C07282=1088.457,205.071,426.735,175.963,20.851,153.236
C07283=1088.452,204.821,426.758,175.960,20.850,153.237
C07284=1088.446,204.573,426.782,175.958,20.848,153.237
C07285=1088.441,204.324,426.805,175.955,20.847,153.237
C07286=1088.435,204.076,426.829,175.952,20.845,153.237
C07287=1088.429,203.827,426.853,175.949,20.844,153.237
C07288=1088.424,203.578,426.877,175.946,20.842,153.237
C07289=1088.418,203.329,426.901,175.944,20.841,153.237
C07290=1088.413,203.080,426.924,175.941,20.839,153.237
C07291=1088.407,202.831,426.948,175.938,20.838,153.238
C07292=1088.402,202.582,426.972,175.936,20.837,153.238
C07293=1088.396,202.334,426.995,175.933,20.836,153.238
C07294=1088.391,202.085,427.019,175.929,20.834,153.238
C07295=1088.385,201.836,427.043,175.927,20.833,153.238
C07296=1088.378,201.587,427.066,175.924,20.831,153.238
C07297=1088.373,201.338,427.090,175.922,20.830,153.239
C07298=1088.367,201.089,427.113,175.919,20.829,153.239
C07299=1088.361,200.841,427.137,175.916,20.827,153.239
C07300=1088.356,200.592,427.160,175.914,20.826,153.239
C07301=1088.350,200.344,427.184,175.910,20.824,153.239
C07302=1088.345,200.095,427.207,175.907,20.823,153.239
C07303=1088.340,199.845,427.230,175.905,20.822,153.240
C07304=1088.334,199.597,427.254,175.902,20.820,153.240
C07305=1088.327,199.348,427.277,175.899,20.819,153.240
C07306=1088.322,199.098,427.301,175.897,20.818,153.240
C07307=1088.316,198.850,427.325,175.894,20.816,153.240
C07308=1088.310,198.601,427.348,175.891,20.814,153.240
C07309=1088.305,198.353,427.372,175.888,20.813,153.241
C07310=1088.299,198.104,427.395,175.885,20.812,153.241
C07311=1088.294,197.855,427.418,175.883,20.811,153.241
C07312=1088.289,197.606,427.441,175.880,20.809,153.241
C07313=1088.283,197.357,427.465,175.877,20.808,153.241
C07314=1088.277,197.108,427.488,175.875,20.807,153.241
C07315=1088.272,196.859,427.511,175.872,20.805,153.241
C07316=1088.266,196.611,427.535,175.870,20.804,153.241
C07317=1088.260,196.362,427.558,175.866,20.802,153.242
C07318=1088.254,196.113,427.581,175.863,20.801,153.242
C07319=1088.249,195.864,427.604,175.861,20.800,153.242
C07320=1088.244,195.615,427.627,175.858,20.798,153.242
C07321=1088.238,195.367,427.651,175.856,20.797,153.242
C07322=1088.233,195.118,427.675,175.853,20.795,153.242
C07323=1088.227,194.869,427.698,175.850,20.794,153.243
C07324=1088.221,194.620,427.721,175.848,20.793,153.243
C07325=1088.216,194.371,427.743,175.845,20.791,153.243
C07326=1088.211,194.122,427.767,175.842,20.790,153.243
C07327=1088.205,193.873,427.791,175.840,20.788,153.243
C07328=1088.199,193.624,427.814,175.836,20.787,153.243
C07329=1088.193,193.376,427.837,175.834,20.786,153.243
C07330=1088.187,193.127,427.859,175.831,20.784,153.244
C07331=1088.182,192.877,427.883,175.828,20.783,153.244
C07332=1088.177,192.629,427.906,175.826,20.781,153.244
C07333=1088.171,192.380,427.929,175.823,20.780,153.244
C07334=1088.165,192.103,427.954,175.821,20.778,153.244
C07335=1088.159,191.825,427.981,175.817,20.777,153.244
C07336=1088.153,191.548,428.006,175.814,20.775,153.244
C07337=1088.146,191.270,428.032,175.811,20.774,153.245
C07338=1088.141,191.021,428.055,175.808,20.772,153.245
C07339=1088.135,190.772,428.078,175.806,20.771,153.245
C07340=1088.130,190.523,428.101,175.803,20.769,153.245
C07341=1088.125,190.275,428.124,175.801,20.768,153.245
C07342=1088.119,190.026,428.147,175.798,20.766,153.245
C07343=1088.113,189.777,428.169,175.795,20.765,153.245
C07344=1088.108,189.528,428.193,175.793,20.763,153.245
C07345=1088.102,189.279,428.216,175.790,20.762,153.246
C07346=1088.097,189.030,428.239,175.787,20.761,153.246
C07347=1088.091,188.782,428.261,175.785,20.760,153.246
C07348=1088.086,188.533,428.284,175.782,20.758,153.246
C07349=1088.080,188.284,428.307,175.780,20.757,153.246
C07350=1088.075,188.035,428.330,175.777,20.755,153.246
C07351=1088.070,187.786,428.353,175.775,20.754,153.246
C07352=1088.064,187.537,428.376,175.771,20.752,153.246
C07353=1088.059,187.289,428.399,175.768,20.750,153.247
C07354=1088.053,187.040,428.422,175.766,20.749,153.247
C07355=1088.048,186.790,428.444,175.763,20.748,153.247
C07356=1088.042,186.541,428.467,175.761,20.746,153.247
C07357=1088.037,186.293,428.489,175.758,20.745,153.247
C07358=1088.031,186.044,428.512,175.756,20.743,153.247
C07359=1088.025,185.795,428.535,175.753,20.742,153.247
C07360=1088.021,185.545,428.558,175.750,20.740,153.247
C07361=1088.015,185.297,428.581,175.748,20.739,153.247
C07362=1088.010,185.048,428.604,175.745,20.737,153.248
C07363=1088.003,184.800,428.626,175.743,20.736,153.248
C07364=1087.998,184.550,428.648,175.740,20.735,153.248
C07365=1087.992,184.301,428.671,175.737,20.734,153.248
C07366=1087.986,184.053,428.694,175.735,20.732,153.248
C07367=1087.981,183.803,428.716,175.732,20.731,153.248
C07368=1087.974,183.554,428.739,175.729,20.729,153.248
C07369=1087.969,183.306,428.761,175.727,20.728,153.249
C07370=1087.964,183.057,428.783,175.724,20.727,153.249
C07371=1087.958,182.808,428.806,175.722,20.725,153.249
C07372=1087.952,182.559,428.829,175.719,20.724,153.249
C07373=1087.946,182.310,428.851,175.716,20.722,153.249
C07374=1087.941,182.061,428.874,175.714,20.722,153.249
C07375=1087.935,181.813,428.896,175.711,20.720,153.249
C07376=1087.929,181.563,428.918,175.708,20.719,153.250
C07377=1087.924,181.315,428.941,175.706,20.717,153.250
C07378=1087.918,181.065,428.963,175.703,20.716,153.250
C07379=1087.912,180.816,428.986,175.701,20.714,153.250
C07380=1087.907,180.568,429.008,175.698,20.713,153.250
C07381=1087.901,180.319,429.031,175.695,20.712,153.250
C07382=1087.895,180.070,429.053,175.693,20.710,153.250
C07383=1087.889,179.821,429.075,175.690,20.709,153.251
C07384=1087.884,179.572,429.098,175.687,20.708,153.251
C07385=1087.878,179.323,429.119,175.685,20.706,153.251
C07386=1087.872,179.074,429.142,175.682,20.705,153.251
C07387=1087.867,178.825,429.164,175.680,20.703,153.251
C07388=1087.861,178.576,429.186,175.677,20.702,153.251
C07389=1087.855,178.327,429.209,175.675,20.700,153.251
C07390=1087.850,178.078,429.231,175.672,20.699,153.252
C07391=1087.844,177.829,429.253,175.669,20.698,153.252
C07392=1087.839,177.580,429.275,175.667,20.696,153.252
C07393=1087.833,177.332,429.298,175.664,20.695,153.252
C07394=1087.827,177.082,429.320,175.661,20.694,153.252
C07395=1087.822,176.834,429.342,175.659,20.692,153.252
C07396=1087.816,176.585,429.365,175.656,20.691,153.252
C07397=1087.810,176.335,429.386,175.654,20.689,153.252
C07398=1087.804,176.058,429.411,175.651,20.688,153.252
C07399=1087.798,175.780,429.436,175.648,20.686,153.253
C07400=1087.792,175.502,429.461,175.645,20.684,153.253
C07401=1087.785,175.225,429.485,175.642,20.683,153.253
C07402=1087.780,174.976,429.507,175.640,20.682,153.253
C07403=1087.774,174.727,429.529,175.637,20.680,153.253
C07404=1087.768,174.477,429.551,175.635,20.679,153.253
C07405=1087.763,174.229,429.574,175.632,20.677,153.253
C07406=1087.757,173.980,429.595,175.630,20.676,153.253
C07407=1087.752,173.731,429.617,175.627,20.674,153.254
C07408=1087.746,173.482,429.639,175.624,20.673,153.254
C07409=1087.740,173.233,429.662,175.623,20.672,153.254
C07410=1087.736,172.984,429.684,175.620,20.670,153.254
C07411=1087.729,172.735,429.705,175.617,20.669,153.254
C07412=1087.724,172.486,429.728,175.615,20.668,153.254
C07413=1087.718,172.238,429.750,175.612,20.666,153.254
C07414=1087.713,171.988,429.772,175.610,20.665,153.254
C07415=1087.707,171.740,429.793,175.607,20.663,153.254
C07416=1087.702,171.490,429.815,175.605,20.662,153.255
C07417=1087.696,171.242,429.837,175.602,20.660,153.255
C07418=1087.691,170.992,429.859,175.600,20.658,153.255
C07419=1087.685,170.743,429.881,175.597,20.657,153.255
C07420=1087.679,170.495,429.903,175.594,20.655,153.255
C07421=1087.674,170.245,429.925,175.592,20.654,153.255
C07422=1087.668,169.997,429.947,175.589,20.653,153.255
C07423=1087.663,169.747,429.969,175.587,20.651,153.255
C07424=1087.657,169.499,429.990,175.584,20.650,153.255
C07425=1087.652,169.249,430.012,175.582,20.649,153.255
C07426=1087.646,169.001,430.034,175.580,20.647,153.256
C07427=1087.641,168.751,430.056,175.577,20.645,153.256
C07428=1087.635,168.503,430.077,175.575,20.644,153.256
C07429=1087.630,168.253,430.099,175.572,20.642,153.256
C07430=1087.624,168.005,430.121,175.570,20.641,153.256
C07431=1087.619,167.755,430.143,175.567,20.640,153.256
C07432=1087.613,167.507,430.164,175.564,20.638,153.256
C07433=1087.608,167.257,430.186,175.562,20.637,153.256
C07434=1087.603,167.009,430.208,175.560,20.635,153.256
C07435=1087.597,166.759,430.230,175.557,20.633,153.256
C07436=1087.592,166.511,430.251,175.554,20.632,153.257
C07437=1087.587,166.262,430.273,175.553,20.631,153.257
C07438=1087.581,166.012,430.295,175.550,20.629,153.257
C07439=1087.575,165.764,430.316,175.548,20.627,153.257
C07440=1087.570,165.514,430.338,175.545,20.626,153.257
C07441=1087.564,165.266,430.359,175.543,20.625,153.257
C07442=1087.559,165.016,430.382,175.540,20.623,153.257
C07443=1087.553,164.767,430.402,175.537,20.622,153.257
C07444=1087.548,164.519,430.424,175.535,20.620,153.257
C07445=1087.542,164.269,430.446,175.532,20.618,153.257
C07446=1087.537,164.021,430.467,175.530,20.617,153.257
C07447=1087.531,163.771,430.489,175.528,20.616,153.257
C07448=1087.526,163.523,430.510,175.526,20.614,153.257
C07449=1087.521,163.274,430.532,175.523,20.613,153.258
C07450=1087.515,163.024,430.553,175.521,20.611,153.258
C07451=1087.510,162.775,430.575,175.518,20.610,153.258
C07452=1087.505,162.527,430.596,175.516,20.608,153.258
C07453=1087.499,162.278,430.618,175.513,20.606,153.258
C07454=1087.494,162.028,430.639,175.510,20.605,153.258
C07455=1087.488,161.779,430.661,175.509,20.603,153.258
C07456=1087.482,161.530,430.682,175.506,20.602,153.258
C07457=1087.477,161.282,430.704,175.504,20.600,153.258
C07458=1087.472,161.032,430.725,175.501,20.599,153.258
C07459=1087.466,160.783,430.746,175.499,20.598,153.258
C07460=1087.460,160.534,430.768,175.496,20.596,153.258
C07461=1087.454,160.286,430.789,175.494,20.594,153.259
C07462=1087.449,160.007,430.813,175.491,20.593,153.259
C07463=1087.442,159.729,430.836,175.489,20.591,153.259
C07464=1087.436,159.451,430.860,175.486,20.590,153.259
C07465=1087.429,159.173,430.883,175.483,20.588,153.259
C07466=1087.424,158.924,430.905,175.481,20.586,153.259
C07467=1087.419,158.675,430.926,175.478,20.585,153.259
C07468=1087.413,158.425,430.948,175.476,20.584,153.259
C07469=1087.407,158.177,430.969,175.473,20.582,153.259
C07470=1087.402,157.928,430.989,175.471,20.580,153.259
C07471=1087.396,157.679,431.011,175.468,20.579,153.260
C07472=1087.390,157.430,431.032,175.467,20.578,153.260
C07473=1087.385,157.181,431.053,175.464,20.576,153.260
C07474=1087.379,156.932,431.074,175.461,20.575,153.260
C07475=1087.374,156.683,431.095,175.459,20.573,153.260
C07476=1087.368,156.434,431.116,175.456,20.571,153.260
C07477=1087.363,156.184,431.138,175.454,20.570,153.260
C07478=1087.357,155.936,431.159,175.452,20.568,153.260
C07479=1087.352,155.686,431.180,175.450,20.567,153.260
C07480=1087.346,155.437,431.201,175.447,20.566,153.260
C07481=1087.341,155.188,431.222,175.445,20.564,153.260
C07482=1087.335,154.940,431.243,175.442,20.562,153.260
C07483=1087.329,154.690,431.264,175.440,20.561,153.260
C07484=1087.324,154.441,431.285,175.437,20.559,153.261
C07485=1087.318,154.192,431.306,175.435,20.558,153.261
C07486=1087.312,153.943,431.327,175.433,20.556,153.261
C07487=1087.306,153.694,431.347,175.430,20.555,153.261
C07488=1087.301,153.445,431.368,175.428,20.554,153.261
C07489=1087.295,153.196,431.390,175.425,20.552,153.261
C07490=1087.290,152.947,431.410,175.423,20.550,153.261
C07491=1087.284,152.698,431.431,175.421,20.549,153.261
C07492=1087.279,152.449,431.452,175.419,20.548,153.261
C07493=1087.273,152.199,431.473,175.416,20.546,153.261
C07494=1087.267,151.951,431.494,175.414,20.544,153.261
C07495=1087.262,151.702,431.515,175.411,20.543,153.261
C07496=1087.257,151.452,431.535,175.410,20.541,153.261
C07497=1087.251,151.203,431.557,175.407,20.540,153.262
C07498=1087.245,150.954,431.577,175.404,20.539,153.262
C07499=1087.240,150.705,431.598,175.402,20.537,153.262
C07500=1087.235,150.456,431.619,175.399,20.535,153.262
C07501=1087.228,150.207,431.640,175.397,20.534,153.262
C07502=1087.223,149.958,431.660,175.395,20.532,153.262
C07503=1087.217,149.709,431.681,175.393,20.531,153.262
C07504=1087.212,149.460,431.702,175.390,20.529,153.262
C07505=1087.206,149.210,431.723,175.388,20.527,153.262
C07506=1087.201,148.961,431.743,175.385,20.526,153.262
C07507=1087.195,148.713,431.765,175.384,20.525,153.262
C07508=1087.189,148.464,431.785,175.381,20.523,153.262
C07509=1087.184,148.215,431.805,175.379,20.522,153.262
C07510=1087.178,147.965,431.826,175.376,20.520,153.262
C07511=1087.173,147.716,431.847,175.374,20.518,153.262
C07512=1087.167,147.468,431.867,175.372,20.517,153.263
C07513=1087.161,147.219,431.888,175.369,20.516,153.263
C07514=1087.156,146.969,431.909,175.367,20.514,153.263
C07515=1087.150,146.720,431.929,175.364,20.512,153.263
C07516=1087.144,146.471,431.949,175.362,20.511,153.263
C07517=1087.139,146.222,431.970,175.360,20.509,153.263
C07518=1087.134,145.973,431.990,175.358,20.508,153.263
C07519=1087.127,145.724,432.011,175.355,20.506,153.263
C07520=1087.122,145.475,432.032,175.353,20.505,153.263
C07521=1087.116,145.225,432.053,175.351,20.504,153.263
C07522=1087.111,144.976,432.073,175.349,20.502,153.263
C07523=1087.105,144.727,432.093,175.346,20.500,153.263
C07524=1087.100,144.478,432.114,175.344,20.498,153.263
C07525=1087.094,144.229,432.135,175.341,20.497,153.263
C07526=1087.087,143.951,432.157,175.339,20.495,153.264
C07527=1087.081,143.672,432.180,175.336,20.493,153.264
C07528=1087.075,143.394,432.203,175.334,20.492,153.264
C07529=1087.069,143.116,432.226,175.331,20.490,153.264
C07530=1087.064,142.867,432.246,175.329,20.489,153.264
C07531=1087.057,142.618,432.267,175.327,20.487,153.264
C07532=1087.052,142.368,432.286,175.325,20.486,153.264
C07533=1087.047,142.119,432.307,175.322,20.484,153.264
C07534=1087.041,141.870,432.327,175.320,20.482,153.264
C07535=1087.036,141.621,432.348,175.317,20.480,153.264
C07536=1087.030,141.372,432.368,175.316,20.479,153.264
C07537=1087.025,141.123,432.388,175.313,20.477,153.264
C07538=1087.019,140.874,432.409,175.311,20.476,153.264
C07539=1087.013,140.625,432.429,175.308,20.474,153.264
C07540=1087.008,140.376,432.449,175.307,20.473,153.264
C07541=1087.001,140.126,432.469,175.304,20.471,153.264
C07542=1086.996,139.877,432.490,175.302,20.470,153.264
C07543=1086.990,139.628,432.510,175.299,20.468,153.264
C07544=1086.985,139.379,432.530,175.298,20.467,153.264
C07545=1086.980,139.129,432.550,175.295,20.465,153.264
C07546=1086.974,138.881,432.570,175.293,20.463,153.264
C07547=1086.969,138.632,432.591,175.290,20.461,153.264
C07548=1086.963,138.383,432.611,175.289,20.460,153.265
C07549=1086.957,138.134,432.631,175.286,20.459,153.265
C07550=1086.952,137.884,432.651,175.284,20.457,153.265
C07551=1086.946,137.635,432.671,175.281,20.455,153.265
C07552=1086.941,137.386,432.691,175.280,20.454,153.265
C07553=1086.935,137.137,432.711,175.277,20.452,153.265
C07554=1086.929,136.888,432.732,175.275,20.451,153.265
C07555=1086.924,136.639,432.751,175.272,20.449,153.265
C07556=1086.918,136.389,432.772,175.271,20.448,153.265
C07557=1086.912,136.140,432.792,175.268,20.446,153.265
C07558=1086.906,135.891,432.812,175.266,20.444,153.265
C07559=1086.901,135.642,432.832,175.264,20.443,153.265
C07560=1086.895,135.393,432.852,175.262,20.442,153.265
C07561=1086.890,135.144,432.872,175.259,20.440,153.265
C07562=1086.884,134.894,432.891,175.257,20.438,153.265
C07563=1086.879,134.645,432.912,175.255,20.437,153.265
C07564=1086.873,134.396,432.932,175.253,20.435,153.265
C07565=1086.867,134.147,432.951,175.250,20.433,153.265
C07566=1086.862,133.898,432.972,175.248,20.431,153.265
C07567=1086.856,133.649,432.992,175.246,20.430,153.265
C07568=1086.851,133.399,433.011,175.244,20.428,153.265
C07569=1086.845,133.150,433.031,175.241,20.427,153.265
C07570=1086.839,132.902,433.051,175.240,20.425,153.265
C07571=1086.834,132.653,433.071,175.237,20.424,153.265
C07572=1086.828,132.404,433.091,175.235,20.422,153.266
C07573=1086.823,132.154,433.110,175.232,20.420,153.266
C07574=1086.817,131.905,433.131,175.231,20.419,153.266
C07575=1086.811,131.656,433.151,175.228,20.417,153.266
C07576=1086.806,131.407,433.170,175.226,20.416,153.266
C07577=1086.800,131.158,433.190,175.224,20.414,153.266
C07578=1086.794,130.909,433.209,175.222,20.412,153.266
C07579=1086.789,130.660,433.230,175.219,20.411,153.266
C07580=1086.783,130.410,433.249,175.217,20.409,153.266
C07581=1086.777,130.161,433.269,175.215,20.408,153.266
C07582=1086.771,129.912,433.288,175.213,20.406,153.266
C07583=1086.765,129.663,433.308,175.210,20.405,153.266
C07584=1086.760,129.414,433.327,175.209,20.403,153.266
C07585=1086.755,129.165,433.348,175.206,20.401,153.266
C07586=1086.749,128.915,433.367,175.204,20.400,153.266
C07587=1086.743,128.666,433.387,175.202,20.398,153.266
C07588=1086.737,128.417,433.406,175.200,20.397,153.266
C07589=1086.731,128.167,433.425,175.197,20.395,153.266
C07590=1086.725,127.889,433.447,175.195,20.393,153.266
C07591=1086.719,127.611,433.470,175.192,20.391,153.266
C07592=1086.713,127.332,433.491,175.190,20.389,153.266
C07593=1086.706,127.054,433.513,175.188,20.388,153.266
C07594=1086.700,126.805,433.533,175.185,20.386,153.266
C07595=1086.694,126.556,433.552,175.184,20.385,153.266
C07596=1086.689,126.306,433.572,175.181,20.383,153.266
C07597=1086.683,126.057,433.592,175.179,20.381,153.266
C07598=1086.678,125.808,433.612,175.177,20.380,153.266
C07599=1086.673,125.559,433.630,175.175,20.378,153.266
C07600=1086.667,125.310,433.650,175.172,20.376,153.266
C07601=1086.661,125.061,433.670,175.171,20.375,153.266
C07602=1086.655,124.811,433.689,175.168,20.373,153.266
C07603=1086.649,124.563,433.709,175.166,20.371,153.267
C07604=1086.644,124.313,433.728,175.164,20.370,153.266
C07605=1086.638,124.064,433.747,175.162,20.368,153.266
C07606=1086.633,123.815,433.766,175.160,20.366,153.266
C07607=1086.627,123.566,433.786,175.158,20.365,153.267
C07608=1086.621,123.317,433.805,175.156,20.363,153.267
C07609=1086.615,123.067,433.825,175.153,20.361,153.267
C07610=1086.610,122.818,433.844,175.152,20.360,153.266
C07611=1086.604,122.569,433.864,175.149,20.358,153.267
C07612=1086.599,122.320,433.883,175.147,20.356,153.267
C07613=1086.594,122.071,433.903,175.145,20.355,153.267
C07614=1086.588,121.821,433.922,175.143,20.353,153.267
C07615=1086.582,121.572,433.941,175.140,20.351,153.267
C07616=1086.576,121.323,433.961,175.139,20.350,153.267
C07617=1086.571,121.074,433.980,175.137,20.348,153.267
C07618=1086.566,120.825,433.999,175.134,20.346,153.267
C07619=1086.560,120.575,434.018,175.133,20.345,153.267
C07620=1086.554,120.326,434.038,175.130,20.343,153.267
C07621=1086.548,120.076,434.057,175.128,20.341,153.267
C07622=1086.543,119.828,434.076,175.126,20.340,153.267
C07623=1086.537,119.579,434.096,175.124,20.338,153.267
C07624=1086.532,119.329,434.115,175.122,20.336,153.267
C07625=1086.526,119.080,434.134,175.120,20.334,153.267
C07626=1086.521,118.831,434.153,175.118,20.333,153.267
C07627=1086.515,118.582,434.172,175.115,20.331,153.267
C07628=1086.510,118.332,434.192,175.114,20.329,153.267
C07629=1086.504,118.084,434.210,175.111,20.327,153.267
C07630=1086.499,117.834,434.230,175.109,20.326,153.267
C07631=1086.493,117.585,434.249,175.107,20.324,153.267
C07632=1086.487,117.335,434.268,175.105,20.322,153.267
C07633=1086.482,117.087,434.287,175.103,20.321,153.267
C07634=1086.477,116.837,434.306,175.101,20.319,153.267
C07635=1086.471,116.588,434.325,175.099,20.317,153.267
C07636=1086.466,116.339,434.344,175.097,20.316,153.267
C07637=1086.460,116.090,434.364,175.095,20.314,153.267
C07638=1086.454,115.840,434.383,175.092,20.312,153.267
C07639=1086.449,115.592,434.401,175.091,20.310,153.266
C07640=1086.443,115.342,434.420,175.089,20.308,153.266
C07641=1086.437,115.093,434.440,175.086,20.306,153.266
C07642=1086.432,114.844,434.459,175.085,20.305,153.266
C07643=1086.427,114.595,434.478,175.082,20.303,153.266
C07644=1086.421,114.345,434.497,175.080,20.301,153.266
C07645=1086.416,114.097,434.516,175.079,20.300,153.266
C07646=1086.410,113.846,434.534,175.076,20.298,153.266
C07647=1086.404,113.597,434.553,175.075,20.297,153.266
C07648=1086.398,113.348,434.572,175.072,20.295,153.266
C07649=1086.393,113.099,434.591,175.070,20.293,153.266
C07650=1086.387,112.850,434.610,175.068,20.291,153.266
C07651=1086.381,112.601,434.629,175.066,20.289,153.266
C07652=1086.376,112.352,434.648,175.064,20.287,153.266
C07653=1086.371,112.102,434.666,175.062,20.286,153.266
C07654=1086.364,111.824,434.688,175.060,20.284,153.266
C07655=1086.358,111.545,434.709,175.057,20.282,153.266
C07656=1086.351,111.267,434.730,175.055,20.280,153.266
C07657=1086.345,110.988,434.751,175.053,20.278,153.266
C07658=1086.340,110.739,434.769,175.050,20.276,153.266
C07659=1086.334,110.490,434.788,175.049,20.275,153.266
C07660=1086.328,110.241,434.807,175.046,20.273,153.266
C07661=1086.322,109.992,434.826,175.045,20.272,153.266
C07662=1086.317,109.742,434.844,175.042,20.270,153.266
C07663=1086.311,109.493,434.863,175.040,20.268,153.266
C07664=1086.305,109.244,434.882,175.039,20.266,153.266
C07665=1086.300,108.995,434.901,175.036,20.264,153.266
C07666=1086.294,108.745,434.919,175.035,20.263,153.266
C07667=1086.288,108.496,434.938,175.032,20.261,153.266
C07668=1086.283,108.247,434.957,175.030,20.259,153.266
C07669=1086.277,107.998,434.975,175.029,20.257,153.266
C07670=1086.271,107.748,434.994,175.026,20.256,153.266
C07671=1086.266,107.499,435.013,175.025,20.254,153.266
C07672=1086.260,107.250,435.031,175.022,20.252,153.266
C07673=1086.255,107.001,435.050,175.020,20.251,153.266
C07674=1086.248,106.751,435.069,175.018,20.249,153.266
C07675=1086.243,106.502,435.087,175.016,20.247,153.266
C07676=1086.237,106.253,435.105,175.014,20.246,153.266
C07677=1086.232,106.004,435.124,175.012,20.244,153.266
C07678=1086.226,105.754,435.143,175.010,20.242,153.266
C07679=1086.221,105.506,435.161,175.008,20.240,153.266
C07680=1086.215,105.256,435.180,175.006,20.238,153.266
C07681=1086.209,105.007,435.198,175.005,20.236,153.266
C07682=1086.204,104.757,435.216,175.002,20.234,153.266
C07683=1086.198,104.508,435.235,175.000,20.232,153.266
C07684=1086.193,104.259,435.254,174.998,20.231,153.266
C07685=1086.186,104.010,435.272,174.996,20.229,153.266
C07686=1086.181,103.761,435.291,174.995,20.228,153.266
C07687=1086.176,103.511,435.309,174.992,20.226,153.266
C07688=1086.170,103.262,435.328,174.990,20.224,153.266
C07689=1086.165,103.012,435.346,174.988,20.222,153.266
C07690=1086.159,102.764,435.364,174.986,20.220,153.266
C07691=1086.154,102.514,435.383,174.985,20.219,153.266
C07692=1086.148,102.265,435.401,174.982,20.217,153.266
C07693=1086.142,102.015,435.420,174.981,20.215,153.266
C07694=1086.136,101.767,435.438,174.978,20.213,153.266
C07695=1086.131,101.517,435.456,174.976,20.211,153.266
C07696=1086.126,101.268,435.474,174.975,20.209,153.265
C07697=1086.120,101.018,435.493,174.972,20.207,153.265
C07698=1086.114,100.769,435.511,174.971,20.206,153.265
C07699=1086.108,100.520,435.529,174.969,20.204,153.265
C07700=1086.103,100.270,435.548,174.966,20.202,153.265
C07701=1086.097,100.021,435.566,174.965,20.201,153.265
C07702=1086.091,99.772,435.584,174.962,20.199,153.265
C07703=1086.086,99.523,435.602,174.961,20.197,153.265
C07704=1086.079,99.274,435.621,174.959,20.195,153.265
C07705=1086.074,99.025,435.639,174.957,20.194,153.265
C07706=1086.069,98.775,435.657,174.955,20.192,153.265
C07707=1086.063,98.526,435.675,174.953,20.190,153.265
C07708=1086.057,98.276,435.693,174.951,20.188,153.265
C07709=1086.052,98.027,435.712,174.949,20.186,153.265
C07710=1086.045,97.778,435.730,174.947,20.185,153.265
C07711=1086.040,97.529,435.748,174.945,20.183,153.265
C07712=1086.034,97.280,435.765,174.943,20.181,153.265
C07713=1086.029,97.030,435.785,174.941,20.179,153.265
C07714=1086.023,96.781,435.802,174.940,20.177,153.265
C07715=1086.017,96.532,435.820,174.937,20.175,153.265
C07716=1086.012,96.282,435.838,174.935,20.173,153.265
C07717=1086.006,96.033,435.857,174.933,20.172,153.265
C07718=1086.000,95.755,435.876,174.931,20.170,153.265
C07719=1085.993,95.477,435.896,174.929,20.168,153.265
C07720=1085.987,95.198,435.918,174.927,20.166,153.265
C07721=1085.981,94.919,435.937,174.925,20.164,153.264
C07722=1085.975,94.671,435.955,174.923,20.162,153.264
C07723=1085.969,94.421,435.973,174.921,20.160,153.264
C07724=1085.964,94.172,435.991,174.919,20.158,153.264
C07725=1085.958,93.922,436.009,174.917,20.156,153.264
C07726=1085.953,93.673,436.027,174.915,20.155,153.264
C07727=1085.947,93.425,436.045,174.913,20.153,153.264
C07728=1085.941,93.175,436.064,174.912,20.151,153.264
C07729=1085.936,92.925,436.081,174.909,20.149,153.264
C07730=1085.930,92.676,436.099,174.908,20.147,153.264
C07731=1085.924,92.427,436.117,174.906,20.145,153.264
C07732=1085.919,92.177,436.135,174.903,20.143,153.264
C07733=1085.913,91.928,436.153,174.902,20.141,153.264
C07734=1085.908,91.679,436.170,174.900,20.139,153.264
C07735=1085.902,91.430,436.188,174.898,20.138,153.264
C07736=1085.896,91.180,436.207,174.896,20.136,153.264
C07737=1085.891,90.931,436.225,174.895,20.134,153.264
C07738=1085.886,90.682,436.242,174.892,20.132,153.264
C07739=1085.879,90.432,436.260,174.891,20.131,153.263
C07740=1085.874,90.183,436.278,174.888,20.129,153.263
C07741=1085.868,89.933,436.296,174.887,20.127,153.263
C07742=1085.862,89.684,436.313,174.885,20.125,153.263
C07743=1085.857,89.435,436.331,174.883,20.123,153.263
C07744=1085.851,89.186,436.349,174.881,20.121,153.263
C07745=1085.845,88.937,436.366,174.879,20.120,153.263
C07746=1085.839,88.687,436.384,174.877,20.118,153.263
C07747=1085.834,88.438,436.402,174.875,20.116,153.263
C07748=1085.828,88.189,436.419,174.873,20.114,153.263
C07749=1085.822,87.939,436.437,174.871,20.112,153.263
C07750=1085.816,87.690,436.455,174.870,20.110,153.263
C07751=1085.811,87.441,436.472,174.867,20.108,153.263
C07752=1085.805,87.191,436.490,174.866,20.106,153.263
C07753=1085.799,86.942,436.508,174.864,20.104,153.263
C07754=1085.794,86.693,436.526,174.862,20.103,153.263
C07755=1085.788,86.443,436.543,174.860,20.101,153.263
C07756=1085.782,86.194,436.560,174.859,20.099,153.262
C07757=1085.777,85.945,436.578,174.856,20.097,153.262
C07758=1085.771,85.695,436.596,174.855,20.096,153.262
C07759=1085.765,85.446,436.613,174.852,20.094,153.262
C07760=1085.760,85.197,436.631,174.851,20.092,153.262
C07761=1085.754,84.948,436.649,174.849,20.090,153.262
C07762=1085.748,84.698,436.666,174.847,20.088,153.262
C07763=1085.743,84.449,436.684,174.845,20.086,153.262
C07764=1085.737,84.199,436.701,174.844,20.084,153.262
C07765=1085.731,83.950,436.719,174.841,20.082,153.262
C07766=1085.726,83.701,436.736,174.840,20.081,153.262
C07767=1085.720,83.452,436.754,174.838,20.078,153.262
C07768=1085.715,83.203,436.772,174.836,20.077,153.262
C07769=1085.708,82.952,436.788,174.834,20.075,153.262
C07770=1085.703,82.703,436.806,174.833,20.073,153.262
C07771=1085.697,82.454,436.823,174.830,20.071,153.262
C07772=1085.692,82.205,436.841,174.829,20.069,153.262
C07773=1085.685,81.956,436.859,174.827,20.067,153.261
C07774=1085.680,81.706,436.876,174.825,20.065,153.261
C07775=1085.675,81.457,436.893,174.823,20.063,153.261
C07776=1085.669,81.208,436.911,174.822,20.061,153.261
C07777=1085.664,80.959,436.928,174.819,20.060,153.261
C07778=1085.658,80.708,436.946,174.818,20.058,153.261
C07779=1085.652,80.459,436.963,174.816,20.056,153.261
C07780=1085.647,80.210,436.981,174.814,20.054,153.261
C07781=1085.641,79.961,436.997,174.812,20.052,153.261
C07782=1085.635,79.683,437.016,174.810,20.050,153.261
C07783=1085.628,79.405,437.037,174.808,20.047,153.261
C07784=1085.622,79.126,437.056,174.806,20.046,153.261
C07785=1085.615,78.848,437.075,174.804,20.043,153.260
C07786=1085.610,78.598,437.092,174.802,20.041,153.260
C07787=1085.605,78.349,437.109,174.801,20.039,153.260
C07788=1085.599,78.099,437.127,174.798,20.037,153.260
C07789=1085.593,77.850,437.144,174.797,20.036,153.260
C07790=1085.587,77.601,437.161,174.795,20.033,153.260
C07791=1085.582,77.352,437.178,174.793,20.032,153.260
C07792=1085.576,77.102,437.195,174.791,20.030,153.260
C07793=1085.570,76.853,437.213,174.790,20.028,153.260
C07794=1085.564,76.603,437.230,174.787,20.026,153.260
C07795=1085.559,76.354,437.247,174.786,20.024,153.260
C07796=1085.554,76.105,437.264,174.784,20.022,153.260
C07797=1085.547,75.856,437.281,174.782,20.020,153.260
C07798=1085.541,75.606,437.299,174.781,20.018,153.259
C07799=1085.536,75.356,437.316,174.779,20.016,153.259
C07800=1085.530,75.108,437.333,174.777,20.015,153.259
C07801=1085.525,74.858,437.350,174.775,20.012,153.259
C07802=1085.519,74.609,437.367,174.773,20.011,153.259
C07803=1085.513,74.360,437.383,174.771,20.009,153.259
C07804=1085.507,74.110,437.401,174.770,20.007,153.259
C07805=1085.502,73.860,437.418,174.767,20.005,153.259
C07806=1085.495,73.612,437.435,174.766,20.003,153.259
C07807=1085.490,73.362,437.452,174.764,20.001,153.259
C07808=1085.485,73.113,437.470,174.763,19.999,153.259
C07809=1085.479,72.864,437.486,174.760,19.997,153.259
C07810=1085.474,72.614,437.503,174.759,19.995,153.258
C07811=1085.468,72.365,437.520,174.757,19.993,153.258
C07812=1085.462,72.115,437.536,174.755,19.992,153.258
C07813=1085.456,71.866,437.554,174.753,19.989,153.258
C07814=1085.451,71.616,437.571,174.752,19.988,153.258
C07815=1085.445,71.367,437.588,174.750,19.985,153.258
C07816=1085.439,71.118,437.605,174.748,19.984,153.258
C07817=1085.433,70.868,437.621,174.747,19.982,153.258
C07818=1085.428,70.619,437.639,174.744,19.980,153.258
C07819=1085.423,70.370,437.656,174.743,19.978,153.258
C07820=1085.417,70.120,437.672,174.741,19.976,153.258
C07821=1085.411,69.871,437.690,174.740,19.974,153.257
C07822=1085.405,69.622,437.706,174.737,19.972,153.257
C07823=1085.400,69.372,437.723,174.736,19.970,153.257
C07824=1085.393,69.123,437.740,174.734,19.968,153.257
C07825=1085.388,68.873,437.757,174.732,19.966,153.257
C07826=1085.382,68.624,437.773,174.730,19.964,153.257
C07827=1085.376,68.375,437.791,174.729,19.962,153.257
C07828=1085.371,68.125,437.807,174.727,19.960,153.257
C07829=1085.365,67.876,437.824,174.725,19.958,153.257
C07830=1085.359,67.627,437.841,174.724,19.956,153.257
C07831=1085.354,67.377,437.858,174.721,19.954,153.257
C07832=1085.348,67.128,437.874,174.720,19.952,153.256
C07833=1085.343,66.878,437.891,174.718,19.950,153.256
C07834=1085.336,66.630,437.908,174.717,19.948,153.256
C07835=1085.331,66.380,437.925,174.714,19.946,153.256
C07836=1085.325,66.131,437.941,174.713,19.944,153.256
C07837=1085.320,65.881,437.958,174.711,19.943,153.256
C07838=1085.314,65.632,437.974,174.709,19.941,153.256
C07839=1085.309,65.383,437.991,174.708,19.939,153.256
C07840=1085.303,65.133,438.008,174.706,19.937,153.256
C07841=1085.297,64.884,438.024,174.704,19.935,153.256
C07842=1085.291,64.634,438.041,174.702,19.933,153.255
C07843=1085.286,64.385,438.057,174.701,19.931,153.255
C07844=1085.279,64.135,438.074,174.699,19.929,153.255
C07845=1085.273,63.886,438.091,174.697,19.927,153.255
C07846=1085.268,63.608,438.109,174.695,19.925,153.255
C07847=1085.261,63.329,438.128,174.693,19.923,153.255
C07848=1085.254,63.051,438.146,174.691,19.921,153.255
C07849=1085.247,62.772,438.165,174.689,19.919,153.255
C07850=1085.241,62.523,438.181,174.688,19.917,153.255
C07851=1085.235,62.274,438.197,174.686,19.915,153.255
C07852=1085.230,62.024,438.214,174.684,19.913,153.255
C07853=1085.224,61.775,438.230,174.682,19.911,153.255
C07854=1085.218,61.525,438.247,174.681,19.909,153.254
C07855=1085.212,61.276,438.263,174.678,19.907,153.254
C07856=1085.207,61.026,438.280,174.677,19.905,153.254
C07857=1085.201,60.777,438.296,174.676,19.903,153.254
C07858=1085.195,60.528,438.312,174.674,19.901,153.254
C07859=1085.189,60.278,438.329,174.672,19.899,153.254
C07860=1085.183,60.029,438.345,174.670,19.897,153.254
C07861=1085.178,59.779,438.362,174.669,19.895,153.254
C07862=1085.172,59.531,438.379,174.666,19.893,153.254
C07863=1085.166,59.281,438.395,174.665,19.891,153.254
C07864=1085.160,59.031,438.410,174.664,19.889,153.253
C07865=1085.154,58.782,438.427,174.661,19.887,153.253
C07866=1085.149,58.532,438.444,174.660,19.885,153.253
C07867=1085.143,58.283,438.460,174.658,19.883,153.253
C07868=1085.137,58.034,438.476,174.657,19.881,153.253
C07869=1085.131,57.784,438.492,174.654,19.879,153.253
C07870=1085.125,57.535,438.509,174.653,19.877,153.253
C07871=1085.119,57.286,438.525,174.651,19.876,153.253
C07872=1085.114,57.036,438.542,174.649,19.873,153.253
C07873=1085.108,56.786,438.558,174.648,19.871,153.252
C07874=1085.102,56.537,438.574,174.646,19.869,153.252
C07875=1085.097,56.289,438.590,174.645,19.867,153.252
C07876=1085.091,56.039,438.606,174.642,19.865,153.252
C07877=1085.085,55.790,438.623,174.641,19.863,153.252
C07878=1085.080,55.540,438.639,174.639,19.862,153.252
C07879=1085.074,55.290,438.655,174.637,19.859,153.252
C07880=1085.068,55.041,438.671,174.636,19.857,153.252
C07881=1085.062,54.791,438.687,174.634,19.855,153.252
C07882=1085.056,54.542,438.704,174.633,19.853,153.252
C07883=1085.050,54.293,438.720,174.631,19.852,153.252
C07884=1085.044,54.043,438.736,174.629,19.849,153.251
C07885=1085.040,53.794,438.752,174.628,19.847,153.251
C07886=1085.034,53.545,438.768,174.625,19.845,153.251
C07887=1085.028,53.295,438.785,174.624,19.843,153.251
C07888=1085.022,53.046,438.801,174.623,19.842,153.251
C07889=1085.016,52.796,438.817,174.621,19.839,153.251
C07890=1085.011,52.546,438.833,174.619,19.837,153.251
C07891=1085.005,52.297,438.849,174.617,19.835,153.251
C07892=1084.999,52.049,438.865,174.616,19.833,153.250
C07893=1084.993,51.799,438.881,174.614,19.831,153.250
C07894=1084.988,51.549,438.897,174.612,19.829,153.250
C07895=1084.983,51.300,438.913,174.611,19.827,153.250
C07896=1084.977,51.050,438.930,174.609,19.825,153.250
C07897=1084.971,50.802,438.946,174.607,19.823,153.250
C07898=1084.966,50.552,438.961,174.605,19.821,153.250
C07899=1084.960,50.302,438.977,174.604,19.819,153.250
C07900=1084.954,50.053,438.994,174.603,19.818,153.250
C07901=1084.948,49.803,439.009,174.600,19.815,153.249
C07902=1084.943,49.554,439.025,174.599,19.813,153.249
C07903=1084.937,49.305,439.041,174.597,19.811,153.249
C07904=1084.931,49.055,439.057,174.596,19.809,153.249
C07905=1084.925,48.806,439.073,174.594,19.807,153.249
C07906=1084.919,48.556,439.089,174.592,19.805,153.249
C07907=1084.914,48.307,439.105,174.591,19.803,153.249
C07908=1084.908,48.058,439.121,174.589,19.801,153.249
C07909=1084.903,47.808,439.138,174.587,19.799,153.249
C07910=1084.897,47.530,439.154,174.585,19.797,153.248
C07911=1084.890,47.251,439.172,174.584,19.795,153.248
C07912=1084.884,46.972,439.190,174.582,19.792,153.248
C07913=1084.878,46.694,439.208,174.580,19.790,153.248
C07914=1084.872,46.444,439.224,174.578,19.788,153.248
C07915=1084.866,46.194,439.240,174.577,19.786,153.248
C07916=1084.861,45.945,439.255,174.575,19.784,153.248
C07917=1084.855,45.696,439.271,174.574,19.782,153.247
C07918=1084.849,45.446,439.288,174.572,19.779,153.247
C07919=1084.844,45.196,439.303,174.570,19.778,153.247
C07920=1084.838,44.948,439.319,174.569,19.776,153.247
C07921=1084.833,44.698,439.334,174.567,19.773,153.247
C07922=1084.827,44.449,439.351,174.565,19.771,153.247
C07923=1084.822,44.199,439.366,174.564,19.770,153.247
C07924=1084.816,43.950,439.382,174.562,19.767,153.246
C07925=1084.810,43.700,439.398,174.561,19.765,153.246
C07926=1084.804,43.451,439.414,174.559,19.763,153.246
C07927=1084.799,43.201,439.429,174.557,19.761,153.246
C07928=1084.793,42.951,439.445,174.556,19.759,153.246
C07929=1084.787,42.702,439.460,174.554,19.757,153.246
C07930=1084.782,42.453,439.476,174.552,19.755,153.246
C07931=1084.776,42.204,439.492,174.550,19.753,153.246
C07932=1084.770,41.954,439.507,174.549,19.751,153.245
C07933=1084.764,41.704,439.524,174.547,19.749,153.245
C07934=1084.758,41.455,439.538,174.545,19.747,153.245
C07935=1084.752,41.206,439.554,174.544,19.744,153.245
C07936=1084.747,40.956,439.570,174.543,19.743,153.245
C07937=1084.742,40.707,439.585,174.541,19.741,153.245
C07938=1084.736,40.458,439.601,174.539,19.738,153.245
C07939=1084.729,40.208,439.616,174.538,19.736,153.245
C07940=1084.724,39.959,439.632,174.536,19.734,153.245
C07941=1084.718,39.709,439.648,174.535,19.732,153.244
C07942=1084.713,39.459,439.663,174.532,19.730,153.244
C07943=1084.708,39.210,439.678,174.531,19.728,153.244
C07944=1084.701,38.961,439.694,174.530,19.726,153.244
C07945=1084.695,38.711,439.710,174.528,19.724,153.244
C07946=1084.690,38.462,439.725,174.526,19.722,153.244
C07947=1084.684,38.212,439.741,174.525,19.720,153.244
C07948=1084.678,37.963,439.756,174.523,19.718,153.243
C07949=1084.673,37.713,439.771,174.522,19.716,153.243
C07950=1084.667,37.464,439.787,174.520,19.713,153.243
C07951=1084.661,37.214,439.802,174.518,19.712,153.243
C07952=1084.655,36.965,439.818,174.517,19.710,153.243
C07953=1084.650,36.715,439.833,174.515,19.707,153.243
C07954=1084.643,36.466,439.849,174.513,19.706,153.243
C07955=1084.638,36.217,439.864,174.512,19.704,153.243
C07956=1084.632,35.967,439.880,174.510,19.701,153.242
C07957=1084.626,35.717,439.894,174.508,19.700,153.242
C07958=1084.621,35.469,439.910,174.507,19.698,153.242
C07959=1084.614,35.219,439.925,174.505,19.695,153.242
C07960=1084.609,34.969,439.941,174.504,19.694,153.242
C07961=1084.604,34.720,439.956,174.502,19.692,153.242
C07962=1084.597,34.471,439.972,174.500,19.689,153.242
C07963=1084.591,34.221,439.987,174.499,19.687,153.242
C07964=1084.586,33.972,440.002,174.498,19.686,153.241
C07965=1084.580,33.722,440.017,174.496,19.683,153.241
C07966=1084.574,33.473,440.032,174.494,19.681,153.241
C07967=1084.568,33.223,440.047,174.492,19.679,153.241
C07968=1084.563,32.974,440.064,174.491,19.677,153.241
C07969=1084.557,32.725,440.078,174.489,19.675,153.241
C07970=1084.551,32.475,440.094,174.487,19.673,153.241
C07971=1084.545,32.226,440.108,174.486,19.671,153.241
C07972=1084.540,31.976,440.124,174.485,19.669,153.240
C07973=1084.533,31.726,440.139,174.483,19.667,153.240
C07974=1084.528,31.447,440.156,174.481,19.665,153.240
C07975=1084.521,31.169,440.173,174.479,19.662,153.240
C07976=1084.514,30.890,440.190,174.478,19.660,153.240
C07977=1084.508,30.612,440.207,174.476,19.658,153.240
C07978=1084.502,30.362,440.222,174.475,19.656,153.239
C07979=1084.497,30.113,440.237,174.472,19.654,153.239
C07980=1084.491,29.863,440.252,174.471,19.652,153.239
C07981=1084.486,29.614,440.267,174.470,19.650,153.239
C07982=1084.479,29.364,440.282,174.468,19.647,153.239
C07983=1084.474,29.115,440.297,174.466,19.646,153.239
C07984=1084.468,28.866,440.313,174.465,19.644,153.239
C07985=1084.462,28.617,440.328,174.463,19.641,153.239
C07986=1084.456,28.367,440.343,174.462,19.639,153.238
C07987=1084.450,28.117,440.359,174.460,19.638,153.238
C07988=1084.445,27.868,440.373,174.458,19.635,153.238
C07989=1084.439,27.618,440.387,174.457,19.633,153.238
C07990=1084.434,27.368,440.403,174.456,19.631,153.238
C07991=1084.427,27.119,440.418,174.453,19.629,153.238
C07992=1084.422,26.869,440.433,174.452,19.627,153.238
C07993=1084.416,26.620,440.448,174.451,19.625,153.238
C07994=1084.410,26.371,440.462,174.449,19.623,153.238
C07995=1084.404,26.121,440.478,174.447,19.621,153.237
C07996=1084.399,25.872,440.492,174.446,19.619,153.237
C07997=1084.393,25.622,440.508,174.444,19.617,153.237
C07998=1084.387,25.373,440.522,174.443,19.615,153.237
C07999=1084.381,25.123,440.537,174.441,19.613,153.237
C08000=1084.376,24.874,440.553,174.439,19.611,153.237
C08001=1084.369,24.624,440.568,174.438,19.609,153.236
C08002=1084.364,24.375,440.581,174.437,19.607,153.236
C08003=1084.358,24.125,440.597,174.435,19.605,153.236
C08004=1084.352,23.876,440.612,174.433,19.603,153.236
C08005=1084.346,23.626,440.626,174.432,19.601,153.236
C08006=1084.341,23.377,440.642,174.430,19.599,153.236
C08007=1084.335,23.127,440.657,174.429,19.597,153.236
C08008=1084.329,22.878,440.671,174.427,19.595,153.236
C08009=1084.323,22.628,440.686,174.425,19.592,153.235
C08010=1084.318,22.379,440.701,174.424,19.591,153.235
C08011=1084.311,22.129,440.716,174.422,19.588,153.235
C08012=1084.305,21.880,440.730,174.421,19.586,153.235
C08013=1084.300,21.630,440.746,174.419,19.584,153.235
C08014=1084.294,21.381,440.760,174.418,19.582,153.235
C08015=1084.288,21.131,440.774,174.416,19.580,153.235
C08016=1084.283,20.882,440.790,174.414,19.578,153.235
C08017=1084.277,20.633,440.804,174.413,19.576,153.234
C08018=1084.271,20.383,440.818,174.412,19.574,153.234
C08019=1084.265,20.134,440.833,174.410,19.572,153.234
C08020=1084.260,19.884,440.849,174.408,19.570,153.234
C08021=1084.254,19.635,440.863,174.407,19.568,153.234
C08022=1084.248,19.384,440.877,174.405,19.565,153.234
C08023=1084.242,19.135,440.892,174.404,19.564,153.234
C08024=1084.236,18.886,440.907,174.402,19.562,153.233
C08025=1084.231,18.636,440.921,174.401,19.560,153.233
C08026=1084.225,18.387,440.936,174.399,19.557,153.233
C08027=1084.219,18.137,440.951,174.398,19.556,153.233
C08028=1084.213,17.888,440.965,174.396,19.554,153.233
C08029=1084.207,17.638,440.980,174.394,19.551,153.233
C08030=1084.202,17.389,440.995,174.393,19.549,153.233
C08031=1084.196,17.139,441.009,174.392,19.548,153.233
C08032=1084.190,16.890,441.024,174.389,19.545,153.232
C08033=1084.184,16.641,441.038,174.388,19.543,153.232
C08034=1084.178,16.390,441.053,174.387,19.541,153.232
C08035=1084.172,16.141,441.067,174.386,19.539,153.232
C08036=1084.167,15.891,441.083,174.383,19.537,153.232
C08037=1084.161,15.642,441.096,174.382,19.535,153.232
C08038=1084.154,15.365,441.113,174.380,19.533,153.232
C08039=1084.148,15.088,441.128,174.379,19.531,153.231
C08040=1084.142,14.811,441.145,174.377,19.528,153.231
C08041=1084.135,14.533,441.160,174.376,19.526,153.231
C08042=1084.130,14.284,441.175,174.374,19.524,153.231
C08043=1084.123,14.035,441.190,174.372,19.522,153.231
C08044=1084.118,13.785,441.204,174.371,19.520,153.231
C08045=1084.111,13.535,441.219,174.370,19.518,153.231
C08046=1084.106,13.286,441.233,174.368,19.516,153.230
C08047=1084.100,13.036,441.248,174.366,19.514,153.230
C08048=1084.094,12.787,441.261,174.365,19.512,153.230
C08049=1084.088,12.538,441.276,174.363,19.509,153.230
C08050=1084.082,12.287,441.290,174.361,19.508,153.230
C08051=1084.076,12.038,441.305,174.360,19.506,153.230
C08052=1084.071,11.789,441.319,174.359,19.504,153.230
C08053=1084.065,11.539,441.334,174.357,19.501,153.230
C08054=1084.059,11.290,441.347,174.355,19.500,153.229
C08055=1084.053,11.040,441.362,174.354,19.498,153.229
C08056=1084.047,10.790,441.376,174.352,19.495,153.229
C08057=1084.041,10.541,441.391,174.351,19.494,153.229
C08058=1084.035,10.291,441.405,174.349,19.492,153.229
C08059=1084.029,10.042,441.418,174.348,19.490,153.229
C08060=1084.023,9.793,441.433,174.346,19.487,153.229
C08061=1084.017,9.543,441.447,174.345,19.486,153.229
C08062=1084.011,9.294,441.462,174.343,19.484,153.228
C08063=1084.006,9.044,441.476,174.341,19.481,153.228
C08064=1084.000,8.794,441.491,174.340,19.479,153.228
C08065=1083.994,8.545,441.504,174.339,19.478,153.228
C08066=1083.989,8.295,441.518,174.337,19.476,153.228
C08067=1083.982,8.046,441.533,174.335,19.473,153.228
C08068=1083.977,7.796,441.547,174.334,19.472,153.228
C08069=1083.971,7.546,441.561,174.333,19.470,153.228
C08070=1083.964,7.297,441.575,174.331,19.468,153.227
C08071=1083.959,7.047,441.589,174.329,19.465,153.227
C08072=1083.953,6.798,441.603,174.328,19.464,153.227
C08073=1083.947,6.549,441.618,174.327,19.462,153.227
C08074=1083.941,6.299,441.632,174.324,19.459,153.227
C08075=1083.936,6.049,441.646,174.323,19.457,153.227
C08076=1083.930,5.800,441.660,174.322,19.456,153.227
C08077=1083.925,5.551,441.674,174.321,19.453,153.226
C08078=1083.918,5.301,441.688,174.319,19.451,153.226
C08079=1083.912,5.052,441.702,174.317,19.449,153.226
C08080=1083.907,4.802,441.716,174.316,19.447,153.226
C08081=1083.901,4.553,441.730,174.315,19.445,153.226
C08082=1083.895,4.302,441.744,174.313,19.443,153.226
C08083=1083.889,4.053,441.759,174.311,19.441,153.226
C08084=1083.884,3.804,441.773,174.310,19.439,153.225
C08085=1083.878,3.554,441.786,174.309,19.437,153.225
C08086=1083.872,3.304,441.800,174.307,19.435,153.225
C08087=1083.866,3.055,441.815,174.305,19.433,153.225
C08088=1083.860,2.806,441.829,174.304,19.431,153.225
C08089=1083.855,2.556,441.843,174.302,19.429,153.225
C08090=1083.849,2.306,441.856,174.301,19.427,153.225
C08091=1083.843,2.056,441.871,174.299,19.425,153.225
C08092=1083.837,1.808,441.885,174.298,19.423,153.224
C08093=1083.831,1.558,441.899,174.296,19.421,153.224
C08094=1083.826,1.308,441.912,174.295,19.419,153.224
C08095=1083.820,1.059,441.926,174.293,19.417,153.224
C08096=1083.814,0.809,441.941,174.292,19.415,153.224
C08097=1083.808,0.559,441.954,174.290,19.412,153.224
C08098=1083.803,0.310,441.968,174.289,19.411,153.224
C08099=1083.797,0.061,441.982,174.287,19.409,153.223
C08100=1083.791,-0.189,441.996,174.286,19.407,153.223
C08101=1083.786,-0.438,442.010,174.284,19.404,153.223
C08102=1083.779,-0.714,442.025,174.283,19.402,153.223
C08103=1083.773,-0.989,442.040,174.281,19.399,153.223
C08104=1083.767,-1.265,442.055,174.280,19.397,153.223
C08105=1083.760,-1.540,442.071,174.277,19.395,153.223
C08106=1083.754,-1.789,442.085,174.276,19.393,153.222
C08107=1083.748,-2.038,442.099,174.275,19.391,153.222
C08108=1083.743,-2.288,442.112,174.274,19.389,153.222
C08109=1083.737,-2.538,442.126,174.272,19.387,153.222
C08110=1083.732,-2.787,442.140,174.270,19.385,153.222
C08111=1083.725,-3.036,442.153,174.269,19.383,153.222
C08112=1083.720,-3.286,442.167,174.268,19.381,153.222
C08113=1083.714,-3.536,442.182,174.266,19.379,153.221
C08114=1083.708,-3.786,442.195,174.264,19.377,153.221
C08115=1083.702,-4.035,442.209,174.263,19.375,153.221
C08116=1083.696,-4.284,442.222,174.262,19.373,153.221
C08117=1083.690,-4.534,442.236,174.260,19.371,153.221
C08118=1083.685,-4.784,442.250,174.258,19.369,153.221
C08119=1083.678,-5.034,442.263,174.257,19.367,153.221
C08120=1083.673,-5.283,442.277,174.256,19.365,153.221
C08121=1083.666,-5.532,442.290,174.254,19.364,153.221
C08122=1083.661,-5.782,442.304,174.252,19.361,153.220
C08123=1083.655,-6.031,442.318,174.251,19.359,153.220
C08124=1083.649,-6.281,442.331,174.249,19.358,153.220
C08125=1083.642,-6.531,442.345,174.248,19.355,153.220
C08126=1083.637,-6.780,442.359,174.246,19.353,153.220
C08127=1083.631,-7.030,442.371,174.245,19.351,153.220
C08128=1083.626,-7.280,442.385,174.243,19.349,153.220
C08129=1083.619,-7.529,442.399,174.242,19.347,153.219
C08130=1083.614,-7.779,442.412,174.240,19.345,153.219
C08131=1083.608,-8.028,442.426,174.239,19.343,153.219
C08132=1083.602,-8.277,442.440,174.238,19.341,153.219
C08133=1083.596,-8.527,442.453,174.236,19.340,153.219
C08134=1083.590,-8.777,442.467,174.234,19.337,153.219
C08135=1083.584,-9.026,442.480,174.233,19.335,153.219
C08136=1083.579,-9.276,442.494,174.232,19.333,153.219
C08137=1083.572,-9.526,442.507,174.230,19.332,153.219
C08138=1083.567,-9.775,442.521,174.229,19.330,153.218
C08139=1083.561,-10.025,442.534,174.227,19.327,153.218
C08140=1083.555,-10.274,442.548,174.225,19.326,153.218
C08141=1083.549,-10.523,442.561,174.224,19.324,153.218
C08142=1083.544,-10.774,442.574,174.223,19.322,153.218
C08143=1083.538,-11.023,442.587,174.221,19.320,153.218
C08144=1083.532,-11.272,442.601,174.219,19.318,153.218
C08145=1083.526,-11.522,442.615,174.218,19.316,153.217
C08146=1083.520,-11.771,442.628,174.217,19.314,153.217
C08147=1083.514,-12.021,442.641,174.215,19.312,153.217
C08148=1083.509,-12.271,442.655,174.213,19.309,153.217
C08149=1083.503,-12.520,442.668,174.212,19.307,153.217
C08150=1083.497,-12.770,442.682,174.211,19.306,153.217
C08151=1083.491,-13.020,442.695,174.210,19.304,153.217
C08152=1083.485,-13.269,442.708,174.207,19.301,153.217
C08153=1083.479,-13.519,442.722,174.206,19.300,153.217
C08154=1083.473,-13.769,442.735,174.205,19.298,153.216
C08155=1083.468,-14.018,442.749,174.204,19.296,153.216
C08156=1083.462,-14.268,442.762,174.202,19.294,153.216
C08157=1083.456,-14.517,442.776,174.200,19.292,153.216
C08158=1083.450,-14.767,442.788,174.199,19.290,153.216
C08159=1083.444,-15.016,442.801,174.198,19.288,153.216
C08160=1083.438,-15.266,442.815,174.196,19.286,153.216
C08161=1083.433,-15.516,442.828,174.195,19.284,153.215
C08162=1083.426,-15.765,442.841,174.193,19.282,153.215
C08163=1083.421,-16.015,442.855,174.191,19.280,153.215
C08164=1083.415,-16.265,442.868,174.190,19.278,153.215
C08165=1083.409,-16.514,442.881,174.189,19.277,153.215
C08166=1083.402,-16.787,442.895,174.187,19.274,153.215
C08167=1083.395,-17.061,442.909,174.185,19.272,153.215
C08168=1083.390,-17.334,442.924,174.183,19.269,153.215
C08169=1083.384,-17.608,442.938,174.182,19.268,153.215
C08170=1083.377,-17.858,442.951,174.181,19.266,153.214
C08171=1083.371,-18.107,442.965,174.180,19.264,153.214
C08172=1083.365,-18.357,442.977,174.177,19.262,153.214
C08173=1083.360,-18.606,442.991,174.176,19.260,153.214
C08174=1083.354,-18.856,443.004,174.175,19.258,153.214
C08175=1083.348,-19.105,443.017,174.173,19.256,153.214
C08176=1083.341,-19.355,443.030,174.172,19.254,153.214
C08177=1083.336,-19.605,443.043,174.170,19.252,153.214
C08178=1083.330,-19.854,443.057,174.169,19.250,153.214
C08179=1083.324,-20.104,443.069,174.167,19.249,153.213
C08180=1083.318,-20.353,443.082,174.166,19.247,153.213
C08181=1083.312,-20.603,443.095,174.165,19.245,153.213
C08182=1083.307,-20.853,443.109,174.162,19.243,153.213
C08183=1083.301,-21.103,443.121,174.161,19.241,153.213
C08184=1083.294,-21.352,443.135,174.160,19.239,153.213
C08185=1083.288,-21.602,443.147,174.159,19.237,153.213
C08186=1083.283,-21.851,443.161,174.157,19.235,153.213
C08187=1083.277,-22.101,443.174,174.155,19.233,153.213
C08188=1083.271,-22.350,443.187,174.154,19.231,153.212
C08189=1083.266,-22.600,443.199,174.153,19.229,153.212
C08190=1083.259,-22.849,443.212,174.151,19.227,153.212
C08191=1083.253,-23.099,443.225,174.150,19.225,153.212
C08192=1083.248,-23.349,443.238,174.148,19.223,153.212
C08193=1083.242,-23.598,443.251,174.146,19.221,153.212
C08194=1083.236,-23.848,443.264,174.145,19.219,153.212
C08195=1083.230,-24.097,443.277,174.144,19.218,153.212
C08196=1083.224,-24.347,443.290,174.142,19.216,153.211
C08197=1083.218,-24.597,443.303,174.141,19.214,153.211
C08198=1083.213,-24.847,443.316,174.139,19.212,153.211
C08199=1083.207,-25.096,443.328,174.138,19.210,153.211
C08200=1083.201,-25.345,443.342,174.136,19.208,153.211
C08201=1083.195,-25.595,443.354,174.135,19.206,153.211
C08202=1083.189,-25.845,443.367,174.134,19.205,153.211
C08203=1083.183,-26.094,443.380,174.132,19.202,153.211
C08204=1083.177,-26.344,443.392,174.130,19.200,153.211
C08205=1083.172,-26.594,443.406,174.129,19.198,153.210
C08206=1083.166,-26.843,443.419,174.128,19.196,153.210
C08207=1083.161,-27.093,443.431,174.126,19.195,153.210
C08208=1083.155,-27.343,443.444,174.125,19.193,153.210
C08209=1083.148,-27.592,443.457,174.123,19.191,153.210
C08210=1083.142,-27.842,443.469,174.122,19.189,153.210
C08211=1083.137,-28.092,443.482,174.120,19.187,153.210
C08212=1083.130,-28.341,443.495,174.119,19.185,153.210
C08213=1083.124,-28.591,443.508,174.117,19.184,153.210
C08214=1083.119,-28.841,443.520,174.116,19.182,153.209
C08215=1083.113,-29.089,443.533,174.114,19.180,153.210
C08216=1083.106,-29.339,443.545,174.113,19.178,153.209
C08217=1083.100,-29.589,443.558,174.111,19.176,153.209
C08218=1083.094,-29.839,443.570,174.110,19.174,153.209
C08219=1083.088,-30.088,443.584,174.109,19.173,153.209
C08220=1083.082,-30.338,443.596,174.107,19.171,153.209
C08221=1083.076,-30.588,443.609,174.105,19.169,153.209
C08222=1083.071,-30.837,443.621,174.104,19.167,153.209
C08223=1083.065,-31.087,443.633,174.102,19.165,153.209
C08224=1083.059,-31.336,443.647,174.101,19.163,153.209
C08225=1083.053,-31.586,443.659,174.100,19.161,153.208
C08226=1083.047,-31.836,443.672,174.099,19.159,153.208
C08227=1083.041,-32.086,443.684,174.096,19.157,153.208
C08228=1083.036,-32.335,443.697,174.095,19.155,153.208
C08229=1083.030,-32.584,443.710,174.094,19.154,153.208
C08230=1083.023,-32.857,443.723,174.092,19.152,153.208
C08231=1083.017,-33.130,443.737,174.090,19.149,153.208
C08232=1083.010,-33.402,443.751,174.089,19.148,153.208
C08233=1083.004,-33.675,443.764,174.088,19.146,153.208
C08234=1082.998,-33.925,443.777,174.085,19.144,153.208
C08235=1082.992,-34.175,443.789,174.084,19.142,153.207
C08236=1082.985,-34.424,443.802,174.083,19.140,153.207
C08237=1082.980,-34.673,443.814,174.081,19.138,153.207
C08238=1082.974,-34.923,443.827,174.080,19.137,153.207
C08239=1082.968,-35.173,443.839,174.079,19.135,153.207
C08240=1082.962,-35.423,443.852,174.077,19.133,153.207
C08241=1082.957,-35.672,443.864,174.075,19.130,153.207
C08242=1082.951,-35.922,443.877,174.074,19.129,153.207
C08243=1082.945,-36.172,443.889,174.073,19.127,153.207
C08244=1082.939,-36.421,443.901,174.071,19.125,153.207
C08245=1082.933,-36.671,443.913,174.070,19.123,153.206
C08246=1082.927,-36.921,443.926,174.069,19.122,153.206
C08247=1082.921,-37.170,443.938,174.066,19.119,153.206
C08248=1082.916,-37.420,443.951,174.065,19.118,153.206
C08249=1082.910,-37.669,443.963,174.064,19.116,153.206
C08250=1082.904,-37.919,443.975,174.062,19.114,153.206
C08251=1082.898,-38.169,443.988,174.061,19.112,153.206
C08252=1082.892,-38.418,444.000,174.060,19.111,153.206
C08253=1082.886,-38.668,444.012,174.058,19.109,153.206
C08254=1082.881,-38.918,444.025,174.056,19.107,153.206
C08255=1082.874,-39.167,444.037,174.055,19.105,153.206
C08256=1082.869,-39.417,444.049,174.054,19.103,153.205
C08257=1082.863,-39.666,444.062,174.052,19.102,153.205
C08258=1082.856,-39.916,444.074,174.051,19.100,153.205
C08259=1082.850,-40.166,444.086,174.049,19.098,153.205
C08260=1082.845,-40.415,444.098,174.048,19.096,153.205
C08261=1082.838,-40.665,444.110,174.047,19.094,153.205
C08262=1082.832,-40.915,444.123,174.044,19.092,153.205
C08263=1082.826,-41.164,444.135,174.043,19.091,153.205
C08264=1082.820,-41.413,444.147,174.042,19.089,153.205
C08265=1082.814,-41.663,444.160,174.040,19.087,153.205
C08266=1082.809,-41.913,444.172,174.039,19.086,153.205
C08267=1082.802,-42.162,444.184,174.038,19.084,153.205
C08268=1082.797,-42.412,444.196,174.036,19.082,153.204
C08269=1082.791,-42.662,444.209,174.035,19.081,153.204
C08270=1082.784,-42.912,444.220,174.033,19.078,153.204
C08271=1082.779,-43.161,444.232,174.031,19.077,153.204
C08272=1082.773,-43.411,444.245,174.030,19.075,153.204
C08273=1082.766,-43.661,444.257,174.029,19.073,153.204
C08274=1082.761,-43.910,444.269,174.027,19.072,153.204
C08275=1082.755,-44.160,444.282,174.026,19.070,153.204
C08276=1082.749,-44.409,444.294,174.025,19.068,153.204
C08277=1082.744,-44.659,444.305,174.023,19.066,153.204
C08278=1082.737,-44.909,444.317,174.021,19.064,153.204
C08279=1082.731,-45.158,444.329,174.020,19.062,153.204
C08280=1082.726,-45.408,444.342,174.018,19.061,153.204
C08281=1082.719,-45.657,444.354,174.017,19.059,153.203
C08282=1082.713,-45.908,444.365,174.015,19.057,153.203
C08283=1082.708,-46.157,444.378,174.014,19.056,153.203
C08284=1082.702,-46.406,444.390,174.013,19.054,153.203
C08285=1082.696,-46.656,444.402,174.011,19.052,153.203
C08286=1082.690,-46.905,444.414,174.009,19.050,153.203
C08287=1082.684,-47.156,444.426,174.008,19.048,153.203
C08288=1082.679,-47.405,444.438,174.006,19.047,153.203
C08289=1082.672,-47.654,444.450,174.005,19.045,153.203
C08290=1082.666,-47.904,444.462,174.004,19.043,153.203
C08291=1082.660,-48.154,444.473,174.002,19.042,153.203
C08292=1082.654,-48.404,444.486,174.001,19.040,153.203
C08293=1082.648,-48.653,444.497,174.000,19.038,153.203
C08294=1082.643,-48.926,444.511,173.997,19.036,153.203
C08295=1082.635,-49.200,444.524,173.996,19.034,153.202
C08296=1082.629,-49.473,444.537,173.995,19.032,153.202
C08297=1082.622,-49.746,444.550,173.993,19.031,153.202
C08298=1082.617,-49.995,444.562,173.991,19.028,153.202
C08299=1082.611,-50.245,444.574,173.990,19.027,153.202
C08300=1082.605,-50.494,444.586,173.988,19.025,153.202
C08301=1082.599,-50.744,444.597,173.987,19.023,153.202
C08302=1082.593,-50.994,444.609,173.986,19.022,153.202
C08303=1082.587,-51.243,444.621,173.984,19.020,153.202
C08304=1082.581,-51.493,444.632,173.983,19.019,153.202
C08305=1082.575,-51.743,444.645,173.981,19.017,153.202
C08306=1082.569,-51.993,444.656,173.980,19.016,153.202
C08307=1082.562,-52.242,444.668,173.979,19.014,153.202
C08308=1082.556,-52.492,444.680,173.976,19.012,153.202
C08309=1082.551,-52.742,444.691,173.975,19.010,153.202
C08310=1082.544,-52.991,444.703,173.973,19.009,153.202
C08311=1082.539,-53.240,444.715,173.972,19.007,153.201
C08312=1082.532,-53.491,444.727,173.971,19.006,153.201
C08313=1082.526,-53.740,444.738,173.969,19.004,153.201
C08314=1082.520,-53.990,444.749,173.968,19.002,153.201
C08315=1082.514,-54.239,444.762,173.966,19.000,153.201
C08316=1082.508,-54.489,444.773,173.965,18.999,153.201
C08317=1082.502,-54.739,444.785,173.964,18.997,153.201
C08318=1082.496,-54.988,444.797,173.962,18.996,153.201
C08319=1082.490,-55.238,444.808,173.961,18.994,153.201
C08320=1082.483,-55.487,444.820,173.959,18.992,153.201
C08321=1082.478,-55.737,444.831,173.957,18.990,153.201
C08322=1082.472,-55.987,444.844,173.956,18.989,153.201
C08323=1082.465,-56.237,444.855,173.954,18.987,153.201
C08324=1082.459,-56.486,444.866,173.953,18.986,153.201
C08325=1082.454,-56.736,444.878,173.951,18.984,153.201
C08326=1082.448,-56.985,444.890,173.950,18.983,153.201
C08327=1082.441,-57.235,444.901,173.948,18.981,153.201
C08328=1082.435,-57.484,444.913,173.947,18.979,153.201
C08329=1082.430,-57.735,444.924,173.946,18.978,153.201
C08330=1082.424,-57.984,444.936,173.944,18.976,153.200
C08331=1082.417,-58.234,444.947,173.943,18.975,153.200
C08332=1082.411,-58.483,444.959,173.941,18.973,153.200
C08333=1082.406,-58.733,444.971,173.940,18.971,153.200
C08334=1082.399,-58.983,444.982,173.939,18.970,153.200
C08335=1082.393,-59.232,444.994,173.936,18.968,153.200
C08336=1082.387,-59.483,445.005,173.935,18.966,153.200
C08337=1082.381,-59.731,445.016,173.934,18.964,153.200
C08338=1082.375,-59.982,445.028,173.932,18.963,153.200
C08339=1082.370,-60.231,445.039,173.931,18.961,153.200
C08340=1082.363,-60.481,445.051,173.929,18.960,153.200
C08341=1082.357,-60.730,445.062,173.928,18.958,153.200
C08342=1082.351,-60.980,445.075,173.926,18.957,153.200
C08343=1082.345,-61.230,445.085,173.925,18.955,153.200
C08344=1082.339,-61.480,445.097,173.924,18.954,153.200
C08345=1082.333,-61.729,445.108,173.922,18.952,153.200
C08346=1082.327,-61.978,445.119,173.921,18.951,153.200
C08347=1082.322,-62.229,445.131,173.919,18.949,153.200
C08348=1082.316,-62.478,445.143,173.918,18.948,153.200
C08349=1082.309,-62.728,445.154,173.917,18.946,153.200
C08350=1082.304,-62.977,445.165,173.915,18.944,153.200
C08351=1082.297,-63.227,445.177,173.914,18.943,153.200
C08352=1082.292,-63.477,445.188,173.911,18.940,153.200
C08353=1082.286,-63.727,445.199,173.910,18.939,153.200
C08354=1082.280,-63.976,445.211,173.908,18.937,153.200
C08355=1082.273,-64.226,445.222,173.907,18.936,153.199
C08356=1082.268,-64.476,445.233,173.906,18.934,153.199
C08357=1082.261,-64.724,445.245,173.904,18.933,153.199
C08358=1082.256,-65.000,445.257,173.903,18.931,153.199
C08359=1082.249,-65.274,445.270,173.901,18.930,153.199
C08360=1082.242,-65.548,445.282,173.900,18.928,153.199
C08361=1082.235,-65.823,445.294,173.898,18.926,153.199
C08362=1082.229,-66.072,445.306,173.896,18.924,153.199
C08363=1082.224,-66.322,445.317,173.895,18.923,153.199
C08364=1082.218,-66.572,445.328,173.893,18.921,153.199
C08365=1082.212,-66.822,445.339,173.892,18.920,153.199
C08366=1082.205,-67.071,445.351,173.891,18.918,153.199
C08367=1082.200,-67.321,445.362,173.889,18.917,153.199
C08368=1082.194,-67.570,445.373,173.888,18.915,153.199
C08369=1082.188,-67.820,445.384,173.886,18.914,153.199
C08370=1082.183,-68.070,445.396,173.885,18.912,153.199
C08371=1082.177,-68.320,445.407,173.883,18.911,153.199
C08372=1082.170,-68.569,445.419,173.882,18.909,153.199
C08373=1082.164,-68.819,445.430,173.880,18.907,153.199
C08374=1082.158,-69.069,445.441,173.879,18.906,153.199
C08375=1082.152,-69.318,445.452,173.878,18.904,153.199
C08376=1082.147,-69.568,445.463,173.876,18.903,153.199
C08377=1082.140,-69.818,445.474,173.875,18.901,153.199
C08378=1082.134,-70.067,445.485,173.873,18.900,153.199
C08379=1082.129,-70.317,445.497,173.872,18.898,153.199
C08380=1082.123,-70.567,445.508,173.870,18.897,153.199
C08381=1082.117,-70.816,445.519,173.869,18.895,153.199
C08382=1082.111,-71.066,445.530,173.867,18.894,153.199
C08383=1082.105,-71.316,445.541,173.866,18.892,153.199
C08384=1082.099,-71.566,445.552,173.865,18.891,153.198
C08385=1082.094,-71.815,445.563,173.863,18.889,153.198
C08386=1082.088,-72.065,445.574,173.862,18.888,153.198
C08387=1082.082,-72.315,445.585,173.860,18.886,153.198
C08388=1082.076,-72.564,445.596,173.859,18.885,153.198
C08389=1082.070,-72.813,445.607,173.857,18.883,153.198
C08390=1082.064,-73.064,445.619,173.856,18.882,153.198
C08391=1082.058,-73.313,445.630,173.853,18.880,153.198
C08392=1082.053,-73.563,445.641,173.852,18.879,153.198
C08393=1082.047,-73.812,445.652,173.850,18.877,153.198
C08394=1082.041,-74.062,445.663,173.849,18.875,153.198
C08395=1082.035,-74.312,445.674,173.848,18.874,153.198
C08396=1082.029,-74.561,445.685,173.846,18.872,153.198
C08397=1082.022,-74.811,445.696,173.845,18.871,153.198
C08398=1082.016,-75.061,445.706,173.843,18.869,153.198
C08399=1082.011,-75.310,445.717,173.842,18.868,153.198
C08400=1082.004,-75.560,445.729,173.840,18.867,153.198
C08401=1081.998,-75.810,445.739,173.839,18.865,153.198
C08402=1081.993,-76.059,445.750,173.837,18.864,153.198
C08403=1081.986,-76.309,445.762,173.836,18.862,153.198
C08404=1081.981,-76.559,445.772,173.834,18.861,153.198
C08405=1081.974,-76.808,445.783,173.833,18.860,153.198
C08406=1081.968,-77.058,445.794,173.832,18.859,153.198
C08407=1081.962,-77.308,445.804,173.831,18.857,153.198
C08408=1081.957,-77.558,445.815,173.829,18.856,153.198
C08409=1081.951,-77.807,445.826,173.828,18.854,153.198
C08410=1081.945,-78.058,445.837,173.826,18.853,153.198
C08411=1081.939,-78.307,445.848,173.825,18.852,153.198
C08412=1081.932,-78.556,445.858,173.823,18.850,153.198
C08413=1081.926,-78.806,445.869,173.822,18.849,153.198
C08414=1081.920,-79.056,445.880,173.820,18.847,153.198
C08415=1081.915,-79.305,445.891,173.818,18.846,153.198
C08416=1081.909,-79.555,445.902,173.817,18.844,153.198
C08417=1081.903,-79.806,445.913,173.816,18.843,153.198
C08418=1081.896,-80.055,445.923,173.814,18.841,153.198
C08419=1081.891,-80.304,445.934,173.812,18.840,153.198
C08420=1081.885,-80.554,445.945,173.811,18.839,153.198
C08421=1081.878,-80.804,445.955,173.810,18.837,153.198
C08422=1081.872,-81.080,445.967,173.808,18.836,153.198
C08423=1081.865,-81.357,445.979,173.806,18.834,153.198
C08424=1081.857,-81.634,445.991,173.804,18.833,153.198
C08425=1081.851,-81.910,446.003,173.803,18.831,153.198
C08426=1081.845,-82.159,446.013,173.801,18.830,153.198
C08427=1081.839,-82.410,446.023,173.800,18.829,153.198
C08428=1081.833,-82.660,446.035,173.798,18.827,153.198
C08429=1081.826,-82.909,446.045,173.796,18.826,153.198
C08430=1081.821,-83.158,446.056,173.795,18.825,153.198
C08431=1081.814,-83.409,446.067,173.794,18.823,153.198
C08432=1081.808,-83.658,446.077,173.792,18.822,153.198
C08433=1081.802,-83.908,446.088,173.790,18.821,153.198
C08434=1081.797,-84.157,446.098,173.789,18.820,153.199
C08435=1081.790,-84.407,446.109,173.787,18.818,153.199
C08436=1081.784,-84.657,446.119,173.786,18.817,153.199
C08437=1081.778,-84.907,446.130,173.785,18.816,153.199
C08438=1081.772,-85.156,446.140,173.784,18.815,153.199
C08439=1081.766,-85.406,446.151,173.782,18.813,153.199
C08440=1081.759,-85.656,446.161,173.780,18.812,153.199
C08441=1081.754,-85.906,446.172,173.779,18.811,153.199
C08442=1081.748,-86.155,446.183,173.777,18.810,153.199
C08443=1081.741,-86.404,446.193,173.776,18.808,153.199
C08444=1081.735,-86.655,446.204,173.774,18.806,153.199
C08445=1081.729,-86.904,446.214,173.773,18.805,153.199
C08446=1081.723,-87.154,446.225,173.771,18.804,153.199
C08447=1081.718,-87.404,446.235,173.770,18.803,153.199
C08448=1081.711,-87.653,446.245,173.768,18.801,153.199
C08449=1081.705,-87.903,446.257,173.766,18.800,153.199
C08450=1081.699,-88.153,446.266,173.765,18.799,153.199
C08451=1081.693,-88.402,446.277,173.764,18.797,153.199
C08452=1081.687,-88.652,446.287,173.762,18.796,153.199
C08453=1081.681,-88.902,446.297,173.760,18.795,153.199
C08454=1081.675,-89.151,446.308,173.759,18.794,153.199
C08455=1081.668,-89.401,446.319,173.758,18.793,153.199
C08456=1081.663,-89.651,446.329,173.756,18.792,153.199
C08457=1081.656,-89.900,446.339,173.755,18.790,153.199
C08458=1081.651,-90.151,446.350,173.754,18.789,153.199
C08459=1081.644,-90.400,446.360,173.752,18.788,153.199
C08460=1081.639,-90.649,446.371,173.750,18.786,153.199
C08461=1081.633,-90.900,446.381,173.749,18.785,153.199
C08462=1081.626,-91.149,446.392,173.747,18.784,153.199
C08463=1081.621,-91.399,446.402,173.746,18.783,153.199
C08464=1081.614,-91.648,446.412,173.744,18.781,153.199
C08465=1081.609,-91.899,446.422,173.742,18.780,153.199
C08466=1081.602,-92.148,446.432,173.741,18.779,153.199
C08467=1081.597,-92.398,446.443,173.739,18.778,153.200
C08468=1081.590,-92.647,446.453,173.738,18.776,153.199
C08469=1081.584,-92.897,446.464,173.737,18.776,153.200
C08470=1081.578,-93.147,446.474,173.736,18.774,153.200
C08471=1081.572,-93.397,446.485,173.734,18.773,153.200
C08472=1081.567,-93.647,446.495,173.732,18.772,153.200
C08473=1081.560,-93.896,446.505,173.731,18.771,153.200
C08474=1081.555,-94.146,446.515,173.729,18.769,153.200
C08475=1081.548,-94.395,446.526,173.728,18.768,153.200
C08476=1081.543,-94.645,446.536,173.726,18.767,153.200
C08477=1081.537,-94.894,446.546,173.725,18.766,153.200
C08478=1081.531,-95.144,446.556,173.723,18.764,153.200
C08479=1081.525,-95.394,446.566,173.721,18.763,153.200
C08480=1081.519,-95.644,446.577,173.720,18.761,153.200
C08481=1081.512,-95.894,446.586,173.719,18.761,153.200
C08482=1081.507,-96.144,446.597,173.717,18.760,153.200
C08483=1081.500,-96.394,446.607,173.716,18.758,153.200
C08484=1081.495,-96.643,446.618,173.714,18.757,153.200
C08485=1081.489,-96.893,446.627,173.713,18.756,153.200
C08486=1081.482,-97.171,446.638,173.711,18.755,153.200
C08487=1081.475,-97.450,446.651,173.710,18.753,153.200
C08488=1081.469,-97.729,446.662,173.708,18.752,153.200
C08489=1081.462,-98.008,446.672,173.706,18.750,153.200
C08490=1081.456,-98.258,446.683,173.705,18.750,153.200
C08491=1081.449,-98.508,446.693,173.703,18.749,153.201
C08492=1081.443,-98.757,446.703,173.702,18.747,153.201
C08493=1081.438,-99.008,446.713,173.700,18.746,153.201
C08494=1081.431,-99.257,446.723,173.698,18.745,153.201
C08495=1081.425,-99.506,446.733,173.697,18.744,153.201
C08496=1081.419,-99.756,446.744,173.695,18.743,153.201
C08497=1081.413,-100.006,446.753,173.694,18.742,153.201
C08498=1081.407,-100.256,446.763,173.692,18.741,153.201
C08499=1081.400,-100.505,446.773,173.691,18.740,153.201
C08500=1081.395,-100.755,446.783,173.690,18.739,153.201
C08501=1081.389,-101.005,446.793,173.688,18.738,153.201
C08502=1081.382,-101.254,446.803,173.686,18.736,153.201
C08503=1081.377,-101.504,446.813,173.685,18.735,153.201
C08504=1081.371,-101.754,446.823,173.683,18.734,153.201
C08505=1081.364,-102.003,446.833,173.681,18.733,153.202
C08506=1081.358,-102.253,446.843,173.680,18.732,153.202
C08507=1081.352,-102.504,446.853,173.679,18.731,153.202
C08508=1081.346,-102.753,446.863,173.677,18.730,153.202
C08509=1081.339,-103.003,446.873,173.676,18.729,153.202
C08510=1081.334,-103.253,446.883,173.674,18.728,153.202
C08511=1081.328,-103.502,446.893,173.673,18.727,153.202
C08512=1081.322,-103.752,446.902,173.671,18.726,153.202
C08513=1081.315,-104.001,446.913,173.669,18.725,153.202
C08514=1081.310,-104.252,446.923,173.669,18.724,153.202
C08515=1081.304,-104.501,446.932,173.667,18.723,153.202
C08516=1081.297,-104.751,446.942,173.665,18.722,153.202
C08517=1081.291,-105.000,446.952,173.664,18.721,153.202
C08518=1081.285,-105.250,446.962,173.662,18.720,153.203
C08519=1081.279,-105.500,446.972,173.660,18.718,153.203
C08520=1081.273,-105.750,446.982,173.659,18.717,153.203
C08521=1081.267,-105.999,446.992,173.657,18.716,153.203
C08522=1081.261,-106.249,447.001,173.656,18.716,153.203
C08523=1081.255,-106.499,447.012,173.654,18.715,153.203
C08524=1081.249,-106.749,447.021,173.653,18.713,153.203
C08525=1081.243,-106.999,447.031,173.651,18.712,153.203
C08526=1081.237,-107.248,447.040,173.650,18.711,153.203
C08527=1081.231,-107.497,447.050,173.648,18.710,153.203
C08528=1081.225,-107.747,447.060,173.647,18.710,153.203
C08529=1081.219,-107.997,447.070,173.645,18.709,153.203
C08530=1081.213,-108.247,447.079,173.644,18.708,153.204
C08531=1081.207,-108.496,447.089,173.642,18.707,153.204
C08532=1081.201,-108.746,447.099,173.641,18.705,153.204
C08533=1081.194,-108.996,447.108,173.639,18.704,153.204
C08534=1081.188,-109.245,447.118,173.637,18.703,153.204
C08535=1081.182,-109.495,447.128,173.636,18.703,153.204
C08536=1081.176,-109.745,447.138,173.635,18.702,153.204
C08537=1081.169,-109.995,447.147,173.633,18.701,153.204
C08538=1081.163,-110.244,447.157,173.631,18.700,153.204
C08539=1081.157,-110.494,447.166,173.630,18.699,153.204
C08540=1081.151,-110.744,447.176,173.628,18.698,153.205
C08541=1081.145,-110.994,447.186,173.627,18.697,153.205
C08542=1081.139,-111.244,447.196,173.625,18.696,153.205
C08543=1081.133,-111.494,447.205,173.624,18.695,153.205
C08544=1081.127,-111.744,447.215,173.622,18.694,153.205
C08545=1081.120,-111.993,447.225,173.620,18.693,153.205
C08546=1081.114,-112.242,447.235,173.619,18.693,153.205
C08547=1081.108,-112.492,447.244,173.618,18.692,153.205
C08548=1081.102,-112.742,447.254,173.616,18.691,153.205
C08549=1081.096,-112.992,447.263,173.614,18.690,153.205
C08550=1081.089,-113.268,447.273,173.613,18.689,153.206
C08551=1081.083,-113.543,447.284,173.611,18.687,153.206
C08552=1081.076,-113.819,447.295,173.610,18.686,153.206
C08553=1081.069,-114.094,447.305,173.608,18.685,153.206
C08554=1081.063,-114.344,447.314,173.606,18.684,153.206
C08555=1081.057,-114.594,447.324,173.604,18.684,153.206
C08556=1081.051,-114.844,447.333,173.603,18.683,153.206
C08557=1081.044,-115.094,447.343,173.602,18.682,153.206
C08558=1081.039,-115.343,447.352,173.600,18.681,153.206
C08559=1081.033,-115.593,447.362,173.598,18.680,153.207
C08560=1081.026,-115.842,447.371,173.597,18.679,153.207
C08561=1081.020,-116.092,447.381,173.596,18.679,153.207
C08562=1081.014,-116.342,447.390,173.594,18.678,153.207
C08563=1081.008,-116.592,447.400,173.592,18.677,153.207
C08564=1081.002,-116.842,447.410,173.591,18.676,153.207
C08565=1080.996,-117.091,447.419,173.589,18.675,153.207
C08566=1080.989,-117.341,447.429,173.588,18.674,153.207
C08567=1080.984,-117.590,447.438,173.586,18.673,153.207
C08568=1080.978,-117.840,447.447,173.585,18.673,153.208
C08569=1080.972,-118.090,447.456,173.583,18.672,153.208
C08570=1080.966,-118.340,447.466,173.581,18.671,153.208
C08571=1080.959,-118.590,447.475,173.580,18.670,153.208
C08572=1080.953,-118.840,447.484,173.579,18.669,153.208
C08573=1080.946,-119.089,447.494,173.577,18.668,153.208
C08574=1080.940,-119.339,447.504,173.575,18.667,153.208
C08575=1080.935,-119.588,447.513,173.574,18.666,153.208
C08576=1080.928,-119.838,447.522,173.572,18.666,153.209
C08577=1080.923,-120.088,447.531,173.571,18.665,153.209
C08578=1080.916,-120.338,447.541,173.569,18.664,153.209
C08579=1080.910,-120.588,447.550,173.567,18.663,153.209
C08580=1080.903,-120.838,447.559,173.566,18.662,153.209
C08581=1080.897,-121.087,447.569,173.565,18.662,153.209
C08582=1080.892,-121.336,447.578,173.563,18.661,153.209
C08583=1080.886,-121.587,447.587,173.561,18.660,153.210
C08584=1080.880,-121.837,447.596,173.559,18.659,153.210
C08585=1080.873,-122.086,447.606,173.559,18.659,153.210
C08586=1080.867,-122.336,447.616,173.557,18.658,153.210
C08587=1080.860,-122.586,447.625,173.555,18.657,153.210
C08588=1080.855,-122.835,447.633,173.553,18.656,153.210
C08589=1080.849,-123.085,447.643,173.552,18.656,153.210
C08590=1080.843,-123.335,447.652,173.551,18.655,153.210
C08591=1080.837,-123.585,447.662,173.549,18.654,153.211
C08592=1080.830,-123.834,447.671,173.547,18.653,153.211
C08593=1080.824,-124.084,447.679,173.545,18.652,153.211
C08594=1080.818,-124.334,447.689,173.545,18.652,153.211
C08595=1080.812,-124.584,447.698,173.543,18.651,153.211
C08596=1080.806,-124.833,447.708,173.541,18.650,153.211
C08597=1080.799,-125.084,447.716,173.539,18.649,153.211
C08598=1080.793,-125.333,447.726,173.538,18.649,153.212
C08599=1080.787,-125.582,447.735,173.536,18.648,153.212
C08600=1080.782,-125.833,447.744,173.535,18.647,153.212
C08601=1080.775,-126.082,447.753,173.533,18.646,153.212
C08602=1080.769,-126.332,447.762,173.532,18.646,153.212
C08603=1080.762,-126.582,447.772,173.530,18.645,153.212
C08604=1080.756,-126.831,447.780,173.529,18.644,153.213
C08605=1080.750,-127.081,447.789,173.527,18.644,153.213
C08606=1080.744,-127.331,447.799,173.526,18.643,153.213
C08607=1080.738,-127.581,447.808,173.524,18.643,153.213
C08608=1080.731,-127.831,447.817,173.522,18.642,153.213
C08609=1080.727,-128.081,447.826,173.521,18.641,153.213
C08610=1080.723,-128.337,447.836,173.519,18.639,153.213
C08611=1080.724,-128.591,447.848,173.518,18.636,153.213
C08612=1080.728,-128.845,447.861,173.518,18.633,153.212
C08613=1080.735,-129.097,447.875,173.518,18.628,153.211
C08614=1080.336,-129.119,447.734,173.474,18.749,153.242
C08615=1080.329,-128.867,447.720,173.474,18.754,153.243
C08616=1080.325,-128.613,447.707,173.474,18.757,153.243
C08617=1080.324,-128.359,447.695,173.475,18.760,153.244
C08618=1080.326,-128.103,447.684,173.476,18.762,153.244
C08619=1080.332,-127.853,447.676,173.478,18.763,153.244
C08620=1080.338,-127.603,447.666,173.480,18.764,153.244
C08621=1080.344,-127.353,447.657,173.482,18.764,153.243
C08622=1080.350,-127.103,447.648,173.483,18.765,153.243
C08623=1080.357,-126.854,447.639,173.484,18.766,153.243
C08624=1080.363,-126.604,447.630,173.486,18.766,153.243
C08625=1080.369,-126.354,447.621,173.488,18.767,153.243
C08626=1080.376,-126.104,447.612,173.489,18.768,153.243
C08627=1080.382,-125.855,447.602,173.491,18.769,153.243
C08628=1080.387,-125.605,447.594,173.492,18.769,153.242
C08629=1080.393,-125.355,447.584,173.494,18.770,153.242
C08630=1080.400,-125.106,447.575,173.495,18.771,153.242
C08631=1080.406,-124.855,447.566,173.497,18.771,153.242
C08632=1080.412,-124.605,447.557,173.499,18.772,153.242
C08633=1080.418,-124.356,447.547,173.500,18.773,153.242
C08634=1080.425,-124.107,447.538,173.501,18.774,153.242
C08635=1080.431,-123.856,447.530,173.503,18.774,153.241
C08636=1080.437,-123.607,447.520,173.505,18.775,153.241
C08637=1080.443,-123.357,447.510,173.507,18.776,153.241
C08638=1080.449,-123.107,447.501,173.508,18.777,153.241
C08639=1080.455,-122.858,447.492,173.509,18.778,153.241
C08640=1080.461,-122.608,447.483,173.511,18.778,153.241
C08641=1080.467,-122.358,447.474,173.513,18.779,153.240
C08642=1080.474,-122.108,447.464,173.514,18.780,153.240
C08643=1080.480,-121.858,447.455,173.515,18.781,153.240
C08644=1080.485,-121.609,447.446,173.517,18.782,153.240
C08645=1080.491,-121.359,447.437,173.519,18.782,153.240
C08646=1080.498,-121.109,447.428,173.521,18.783,153.240
C08647=1080.504,-120.860,447.418,173.522,18.784,153.240
C08648=1080.510,-120.610,447.409,173.523,18.784,153.240
C08649=1080.517,-120.360,447.399,173.525,18.785,153.239
C08650=1080.523,-120.110,447.389,173.527,18.786,153.239
C08651=1080.528,-119.860,447.381,173.528,18.787,153.239
C08652=1080.534,-119.611,447.371,173.529,18.787,153.239
C08653=1080.541,-119.361,447.362,173.531,18.788,153.239
C08654=1080.547,-119.111,447.353,173.533,18.789,153.239
C08655=1080.553,-118.862,447.343,173.534,18.790,153.239
C08656=1080.560,-118.612,447.334,173.536,18.791,153.239
C08657=1080.566,-118.362,447.324,173.537,18.792,153.239
C08658=1080.571,-118.113,447.315,173.539,18.793,153.238
C08659=1080.577,-117.862,447.306,173.540,18.794,153.238
C08660=1080.583,-117.613,447.297,173.542,18.795,153.238
C08661=1080.590,-117.363,447.287,173.544,18.796,153.238
C08662=1080.596,-117.113,447.277,173.545,18.796,153.238
C08663=1080.602,-116.863,447.268,173.547,18.797,153.238
C08664=1080.608,-116.613,447.258,173.548,18.798,153.238
C08665=1080.614,-116.364,447.249,173.550,18.799,153.237
C08666=1080.621,-116.114,447.240,173.552,18.800,153.237
C08667=1080.627,-115.865,447.231,173.553,18.801,153.237
C08668=1080.633,-115.615,447.221,173.554,18.801,153.237
C08669=1080.639,-115.365,447.211,173.556,18.802,153.237
C08670=1080.645,-115.116,447.202,173.558,18.803,153.237
C08671=1080.651,-114.866,447.192,173.559,18.804,153.237
C08672=1080.658,-114.616,447.183,173.561,18.805,153.237
C08673=1080.664,-114.366,447.173,173.562,18.806,153.237
C08674=1080.670,-114.116,447.164,173.563,18.807,153.237
C08675=1080.676,-113.840,447.153,173.565,18.808,153.236
C08676=1080.683,-113.565,447.143,173.567,18.809,153.236
C08677=1080.690,-113.288,447.132,173.569,18.810,153.236
C08678=1080.697,-113.013,447.121,173.570,18.811,153.236
C08679=1080.703,-112.763,447.112,173.572,18.812,153.236
C08680=1080.709,-112.513,447.102,173.574,18.813,153.236
C08681=1080.715,-112.263,447.092,173.575,18.814,153.236
C08682=1080.721,-112.014,447.083,173.577,18.815,153.236
C08683=1080.727,-111.765,447.074,173.578,18.815,153.236
C08684=1080.733,-111.515,447.064,173.579,18.817,153.236
C08685=1080.739,-111.265,447.055,173.581,18.818,153.235
C08686=1080.745,-111.015,447.045,173.583,18.819,153.235
C08687=1080.752,-110.765,447.035,173.584,18.820,153.235
C08688=1080.757,-110.515,447.025,173.586,18.821,153.235
C08689=1080.763,-110.266,447.015,173.587,18.821,153.235
C08690=1080.770,-110.016,447.005,173.589,18.822,153.235
C08691=1080.776,-109.766,446.996,173.590,18.823,153.235
C08692=1080.782,-109.517,446.986,173.592,18.824,153.235
C08693=1080.788,-109.267,446.977,173.594,18.825,153.235
C08694=1080.794,-109.017,446.967,173.595,18.826,153.234
C08695=1080.800,-108.767,446.958,173.596,18.827,153.235
C08696=1080.807,-108.518,446.948,173.598,18.828,153.234
C08697=1080.813,-108.268,446.938,173.599,18.829,153.234
C08698=1080.819,-108.019,446.928,173.601,18.830,153.234
C08699=1080.825,-107.768,446.918,173.603,18.831,153.234
C08700=1080.831,-107.519,446.908,173.604,18.832,153.234
C08701=1080.837,-107.269,446.899,173.606,18.833,153.234
C08702=1080.843,-107.019,446.889,173.607,18.834,153.234
C08703=1080.849,-106.769,446.880,173.608,18.835,153.234
C08704=1080.856,-106.520,446.869,173.610,18.836,153.234
C08705=1080.861,-106.270,446.859,173.612,18.837,153.234
C08706=1080.867,-106.020,446.850,173.614,18.838,153.233
C08707=1080.874,-105.770,446.840,173.615,18.840,153.233
C08708=1080.880,-105.521,446.831,173.617,18.841,153.233
C08709=1080.886,-105.271,446.820,173.618,18.841,153.233
C08710=1080.892,-105.021,446.810,173.619,18.842,153.233
C08711=1080.898,-104.771,446.801,173.621,18.844,153.233
C08712=1080.904,-104.522,446.791,173.622,18.845,153.233
C08713=1080.911,-104.272,446.781,173.624,18.846,153.233
C08714=1080.916,-104.022,446.771,173.626,18.847,153.233
C08715=1080.922,-103.773,446.761,173.627,18.848,153.233
C08716=1080.928,-103.523,446.751,173.629,18.849,153.233
C08717=1080.935,-103.274,446.741,173.630,18.850,153.233
C08718=1080.940,-103.023,446.731,173.631,18.851,153.233
C08719=1080.946,-102.774,446.721,173.633,18.852,153.233
C08720=1080.953,-102.524,446.712,173.635,18.853,153.232
C08721=1080.959,-102.275,446.702,173.636,18.854,153.232
C08722=1080.964,-102.025,446.691,173.638,18.856,153.232
C08723=1080.971,-101.775,446.682,173.639,18.857,153.232
C08724=1080.977,-101.526,446.672,173.641,18.858,153.232
C08725=1080.983,-101.276,446.661,173.642,18.859,153.232
C08726=1080.989,-101.026,446.652,173.643,18.860,153.232
C08727=1080.995,-100.777,446.642,173.645,18.861,153.232
C08728=1081.001,-100.527,446.632,173.647,18.862,153.232
C08729=1081.007,-100.277,446.622,173.648,18.863,153.232
C08730=1081.013,-100.027,446.612,173.650,18.864,153.232
C08731=1081.019,-99.778,446.602,173.652,18.865,153.232
C08732=1081.025,-99.528,446.592,173.653,18.867,153.232
C08733=1081.032,-99.278,446.581,173.655,18.868,153.232
C08734=1081.038,-99.028,446.572,173.656,18.868,153.232
C08735=1081.044,-98.778,446.561,173.657,18.870,153.232
C08736=1081.050,-98.529,446.551,173.659,18.871,153.231
C08737=1081.056,-98.279,446.542,173.660,18.872,153.231
C08738=1081.062,-98.029,446.531,173.662,18.873,153.231
C08739=1081.069,-97.750,446.520,173.664,18.874,153.231
C08740=1081.076,-97.471,446.508,173.665,18.876,153.231
C08741=1081.082,-97.192,446.497,173.667,18.877,153.231
C08742=1081.089,-96.913,446.486,173.668,18.878,153.231
C08743=1081.096,-96.664,446.476,173.670,18.879,153.231
C08744=1081.101,-96.414,446.466,173.671,18.881,153.231
C08745=1081.107,-96.164,446.456,173.673,18.882,153.231
C08746=1081.113,-95.915,446.445,173.674,18.883,153.231
C08747=1081.119,-95.665,446.436,173.676,18.884,153.231
C08748=1081.125,-95.415,446.425,173.678,18.886,153.231
C08749=1081.131,-95.166,446.415,173.679,18.887,153.231
C08750=1081.137,-94.915,446.404,173.681,18.888,153.231
C08751=1081.143,-94.665,446.394,173.682,18.889,153.231
C08752=1081.149,-94.416,446.383,173.684,18.891,153.231
C08753=1081.155,-94.166,446.373,173.686,18.892,153.231
C08754=1081.161,-93.917,446.363,173.686,18.893,153.231
C08755=1081.167,-93.667,446.353,173.688,18.894,153.231
C08756=1081.173,-93.417,446.343,173.689,18.895,153.231
C08757=1081.178,-93.167,446.332,173.691,18.896,153.231
C08758=1081.185,-92.918,446.322,173.692,18.898,153.231
C08759=1081.190,-92.668,446.312,173.694,18.899,153.230
C08760=1081.197,-92.418,446.301,173.696,18.900,153.230
C08761=1081.203,-92.168,446.291,173.697,18.901,153.230
C08762=1081.209,-91.919,446.281,173.699,18.903,153.230
C08763=1081.215,-91.669,446.270,173.700,18.904,153.230
C08764=1081.221,-91.420,446.260,173.702,18.905,153.230
C08765=1081.227,-91.170,446.249,173.703,18.907,153.230
C08766=1081.232,-90.920,446.239,173.705,18.908,153.230
C08767=1081.239,-90.671,446.229,173.706,18.909,153.230
C08768=1081.245,-90.420,446.219,173.707,18.910,153.230
C08769=1081.251,-90.171,446.208,173.709,18.911,153.230
C08770=1081.257,-89.921,446.197,173.711,18.912,153.230
C08771=1081.263,-89.672,446.188,173.712,18.914,153.230
C08772=1081.269,-89.422,446.177,173.713,18.916,153.230
C08773=1081.275,-89.172,446.167,173.715,18.917,153.230
C08774=1081.282,-88.922,446.156,173.717,18.918,153.230
C08775=1081.287,-88.673,446.145,173.718,18.919,153.230
C08776=1081.294,-88.423,446.136,173.720,18.921,153.230
C08777=1081.299,-88.173,446.125,173.721,18.922,153.230
C08778=1081.306,-87.924,446.115,173.723,18.923,153.230
C08779=1081.311,-87.674,446.104,173.724,18.925,153.230
C08780=1081.318,-87.424,446.093,173.726,18.926,153.230
C08781=1081.324,-87.175,446.083,173.727,18.927,153.230
C08782=1081.329,-86.925,446.073,173.729,18.929,153.230
C08783=1081.336,-86.675,446.062,173.731,18.930,153.230
C08784=1081.342,-86.426,446.051,173.732,18.931,153.230
C08785=1081.348,-86.176,446.040,173.733,18.932,153.230
C08786=1081.354,-85.926,446.031,173.734,18.933,153.230
C08787=1081.360,-85.676,446.020,173.736,18.935,153.230
C08788=1081.366,-85.427,446.010,173.737,18.936,153.230
C08789=1081.372,-85.176,445.999,173.739,18.937,153.230
C08790=1081.378,-84.927,445.988,173.740,18.939,153.230
C08791=1081.385,-84.678,445.978,173.742,18.940,153.230
C08792=1081.390,-84.428,445.967,173.743,18.941,153.230
C08793=1081.396,-84.177,445.956,173.745,18.943,153.230
C08794=1081.403,-83.928,445.946,173.747,18.944,153.230
C08795=1081.409,-83.679,445.935,173.748,18.945,153.230
C08796=1081.415,-83.430,445.925,173.750,18.947,153.230
C08797=1081.421,-83.179,445.914,173.751,18.948,153.229
C08798=1081.427,-82.929,445.904,173.753,18.949,153.230
C08799=1081.433,-82.680,445.893,173.754,18.951,153.230
C08800=1081.439,-82.431,445.882,173.756,18.952,153.230
C08801=1081.445,-82.180,445.871,173.757,18.953,153.229
C08802=1081.452,-81.931,445.861,173.759,18.955,153.229
C08803=1081.458,-81.654,445.849,173.760,18.956,153.230
C08804=1081.465,-81.377,445.838,173.762,18.957,153.229
C08805=1081.471,-81.100,445.825,173.763,18.959,153.229
C08806=1081.479,-80.823,445.814,173.766,18.961,153.229
C08807=1081.485,-80.574,445.803,173.767,18.962,153.229
C08808=1081.491,-80.325,445.792,173.769,18.963,153.229
C08809=1081.497,-80.075,445.782,173.769,18.964,153.229
C08810=1081.503,-79.825,445.770,173.771,18.966,153.229
C08811=1081.509,-79.576,445.759,173.772,18.967,153.229
C08812=1081.515,-79.326,445.750,173.774,18.969,153.230
C08813=1081.521,-79.076,445.739,173.775,18.970,153.229
C08814=1081.527,-78.826,445.728,173.777,18.972,153.229
C08815=1081.533,-78.577,445.717,173.778,18.973,153.229
C08816=1081.539,-78.327,445.706,173.780,18.975,153.229
C08817=1081.545,-78.077,445.695,173.781,18.976,153.230
C08818=1081.551,-77.828,445.684,173.783,18.977,153.229
C08819=1081.557,-77.578,445.674,173.784,18.979,153.229
C08820=1081.563,-77.329,445.663,173.786,18.980,153.229
C08821=1081.569,-77.079,445.651,173.787,18.982,153.229
C08822=1081.575,-76.829,445.641,173.789,18.983,153.230
C08823=1081.581,-76.580,445.630,173.790,18.985,153.230
C08824=1081.587,-76.329,445.618,173.792,18.986,153.230
C08825=1081.594,-76.080,445.608,173.793,18.987,153.229
C08826=1081.599,-75.831,445.597,173.795,18.989,153.229
C08827=1081.606,-75.581,445.586,173.796,18.990,153.230
C08828=1081.611,-75.330,445.576,173.798,18.992,153.230
C08829=1081.617,-75.081,445.565,173.799,18.993,153.230
C08830=1081.623,-74.831,445.553,173.801,18.995,153.230
C08831=1081.629,-74.582,445.542,173.802,18.996,153.230
C08832=1081.635,-74.332,445.531,173.803,18.998,153.230
C08833=1081.641,-74.082,445.520,173.805,18.999,153.230
C08834=1081.647,-73.833,445.509,173.807,19.000,153.230
C08835=1081.653,-73.583,445.498,173.808,19.002,153.230
C08836=1081.658,-73.334,445.487,173.809,19.003,153.230
C08837=1081.665,-73.084,445.476,173.811,19.005,153.230
C08838=1081.671,-72.834,445.465,173.812,19.006,153.230
C08839=1081.676,-72.585,445.454,173.814,19.008,153.230
C08840=1081.683,-72.334,445.443,173.815,19.009,153.230
C08841=1081.688,-72.085,445.432,173.817,19.011,153.230
C08842=1081.694,-71.835,445.421,173.818,19.013,153.230
C08843=1081.700,-71.585,445.410,173.820,19.014,153.230
C08844=1081.706,-71.336,445.399,173.822,19.016,153.230
C08845=1081.712,-71.086,445.388,173.823,19.018,153.230
C08846=1081.717,-70.836,445.377,173.825,19.019,153.230
C08847=1081.724,-70.587,445.365,173.826,19.021,153.230
C08848=1081.729,-70.337,445.354,173.828,19.022,153.230
C08849=1081.735,-70.088,445.343,173.829,19.024,153.230
C08850=1081.741,-69.838,445.332,173.830,19.026,153.230
C08851=1081.747,-69.588,445.321,173.832,19.027,153.230
C08852=1081.753,-69.338,445.310,173.833,19.029,153.230
C08853=1081.759,-69.089,445.299,173.835,19.030,153.230
C08854=1081.765,-68.840,445.287,173.836,19.032,153.230
C08855=1081.771,-68.589,445.276,173.838,19.033,153.230
C08856=1081.777,-68.340,445.265,173.839,19.035,153.230
C08857=1081.782,-68.090,445.254,173.841,19.036,153.230
C08858=1081.789,-67.840,445.243,173.842,19.038,153.230
C08859=1081.794,-67.591,445.232,173.843,19.039,153.230
C08860=1081.800,-67.342,445.220,173.845,19.041,153.230
C08861=1081.807,-67.091,445.209,173.846,19.042,153.231
C08862=1081.812,-66.842,445.197,173.848,19.044,153.231
C08863=1081.818,-66.591,445.186,173.849,19.045,153.231
C08864=1081.824,-66.343,445.175,173.851,19.047,153.231
C08865=1081.830,-66.093,445.164,173.852,19.048,153.231
C08866=1081.836,-65.843,445.152,173.854,19.050,153.231
C08867=1081.843,-65.569,445.140,173.855,19.052,153.231
C08868=1081.849,-65.293,445.127,173.857,19.054,153.231
C08869=1081.855,-65.020,445.115,173.859,19.056,153.231
C08870=1081.862,-64.745,445.103,173.860,19.057,153.231
C08871=1081.869,-64.495,445.091,173.861,19.059,153.231
C08872=1081.874,-64.245,445.080,173.863,19.060,153.231
C08873=1081.880,-63.995,445.069,173.864,19.062,153.231
C08874=1081.886,-63.746,445.057,173.866,19.064,153.231
C08875=1081.892,-63.496,445.046,173.867,19.065,153.231
C08876=1081.898,-63.247,445.035,173.869,19.067,153.231
C08877=1081.904,-62.998,445.023,173.871,19.069,153.231
C08878=1081.910,-62.747,445.011,173.872,19.070,153.231
C08879=1081.915,-62.498,445.001,173.874,19.072,153.231
C08880=1081.922,-62.248,444.989,173.875,19.073,153.231
C08881=1081.928,-61.999,444.978,173.877,19.075,153.231
C08882=1081.934,-61.749,444.967,173.878,19.076,153.231
C08883=1081.939,-61.499,444.954,173.879,19.078,153.232
C08884=1081.946,-61.249,444.943,173.881,19.080,153.232
C08885=1081.952,-61.000,444.932,173.882,19.081,153.232
C08886=1081.958,-60.750,444.920,173.884,19.083,153.232
C08887=1081.964,-60.501,444.909,173.885,19.084,153.232
C08888=1081.970,-60.251,444.897,173.887,19.086,153.232
C08889=1081.976,-60.001,444.886,173.888,19.087,153.232
C08890=1081.982,-59.751,444.875,173.889,19.090,153.232
C08891=1081.988,-59.502,444.863,173.891,19.091,153.232
C08892=1081.994,-59.252,444.851,173.892,19.093,153.232
C08893=1082.000,-59.003,444.840,173.894,19.095,153.232
C08894=1082.006,-58.753,444.828,173.896,19.096,153.232
C08895=1082.012,-58.504,444.817,173.897,19.098,153.232
C08896=1082.018,-58.253,444.805,173.899,19.099,153.232
C08897=1082.024,-58.004,444.793,173.900,19.101,153.232
C08898=1082.030,-57.754,444.782,173.901,19.103,153.232
C08899=1082.037,-57.505,444.770,173.903,19.104,153.232
C08900=1082.042,-57.255,444.759,173.904,19.106,153.232
C08901=1082.048,-57.005,444.747,173.906,19.107,153.232
C08902=1082.054,-56.756,444.736,173.907,19.109,153.232
C08903=1082.061,-56.506,444.724,173.908,19.111,153.233
C08904=1082.066,-56.256,444.712,173.910,19.112,153.233
C08905=1082.072,-56.007,444.700,173.911,19.114,153.233
C08906=1082.079,-55.757,444.689,173.913,19.115,153.233
C08907=1082.085,-55.508,444.678,173.915,19.117,153.233
C08908=1082.090,-55.257,444.666,173.917,19.119,153.233
C08909=1082.096,-55.008,444.654,173.918,19.121,153.233
C08910=1082.103,-54.758,444.643,173.919,19.122,153.233
C08911=1082.108,-54.509,444.631,173.921,19.124,153.233
C08912=1082.114,-54.259,444.620,173.922,19.125,153.233
C08913=1082.121,-54.009,444.608,173.924,19.127,153.233
C08914=1082.127,-53.760,444.596,173.925,19.129,153.233
C08915=1082.133,-53.510,444.584,173.926,19.131,153.233
C08916=1082.139,-53.260,444.572,173.928,19.132,153.233
C08917=1082.145,-53.011,444.561,173.929,19.134,153.233
C08918=1082.151,-52.761,444.549,173.931,19.135,153.233
C08919=1082.157,-52.512,444.537,173.933,19.138,153.233
C08920=1082.163,-52.262,444.526,173.934,19.139,153.233
C08921=1082.169,-52.012,444.513,173.936,19.141,153.233
C08922=1082.175,-51.762,444.503,173.937,19.142,153.233
C08923=1082.182,-51.513,444.491,173.938,19.144,153.234
C08924=1082.188,-51.263,444.478,173.940,19.146,153.234
C08925=1082.193,-51.014,444.467,173.941,19.147,153.234
C08926=1082.200,-50.764,444.455,173.943,19.149,153.234
C08927=1082.206,-50.514,444.443,173.944,19.150,153.234
C08928=1082.212,-50.265,444.432,173.945,19.152,153.234
C08929=1082.217,-50.015,444.419,173.947,19.154,153.234
C08930=1082.224,-49.766,444.408,173.949,19.156,153.234
C08931=1082.230,-49.492,444.394,173.950,19.158,153.234
C08932=1082.237,-49.219,444.381,173.952,19.159,153.234
C08933=1082.243,-48.945,444.369,173.953,19.161,153.234
C08934=1082.250,-48.672,444.356,173.955,19.163,153.234
C08935=1082.255,-48.422,444.343,173.956,19.165,153.235
C08936=1082.261,-48.173,444.331,173.958,19.167,153.235
C08937=1082.267,-47.923,444.320,173.959,19.169,153.235
C08938=1082.272,-47.674,444.307,173.961,19.171,153.235
C08939=1082.279,-47.424,444.295,173.962,19.172,153.235
C08940=1082.285,-47.174,444.283,173.963,19.174,153.235
C08941=1082.291,-46.925,444.271,173.966,19.176,153.235
C08942=1082.297,-46.675,444.259,173.967,19.178,153.235
C08943=1082.302,-46.425,444.247,173.968,19.180,153.235
C08944=1082.309,-46.176,444.235,173.970,19.181,153.235
C08945=1082.314,-45.926,444.223,173.971,19.183,153.235
C08946=1082.319,-45.677,444.211,173.972,19.185,153.235
C08947=1082.326,-45.427,444.199,173.974,19.186,153.235
C08948=1082.332,-45.177,444.187,173.975,19.188,153.236
C08949=1082.338,-44.928,444.175,173.976,19.190,153.236
C08950=1082.344,-44.678,444.163,173.979,19.192,153.236
C08951=1082.350,-44.428,444.150,173.980,19.194,153.236
C08952=1082.356,-44.179,444.139,173.981,19.195,153.236
C08953=1082.362,-43.929,444.127,173.983,19.197,153.236
C08954=1082.367,-43.679,444.114,173.984,19.199,153.236
C08955=1082.373,-43.430,444.102,173.986,19.200,153.236
C08956=1082.379,-43.180,444.090,173.987,19.202,153.236
C08957=1082.386,-42.931,444.078,173.988,19.204,153.236
C08958=1082.392,-42.681,444.065,173.990,19.207,153.236
C08959=1082.397,-42.432,444.053,173.992,19.208,153.236
C08960=1082.404,-42.182,444.042,173.993,19.210,153.236
C08961=1082.409,-41.932,444.029,173.994,19.212,153.237
C08962=1082.415,-41.683,444.017,173.996,19.213,153.237
C08963=1082.421,-41.433,444.005,173.997,19.215,153.237
C08964=1082.427,-41.183,443.993,173.999,19.217,153.237
C08965=1082.433,-40.933,443.980,174.000,19.219,153.237
C08966=1082.439,-40.684,443.969,174.002,19.221,153.237
C08967=1082.445,-40.434,443.956,174.003,19.222,153.237
C08968=1082.451,-40.185,443.943,174.005,19.224,153.237
C08969=1082.458,-39.935,443.932,174.006,19.226,153.237
C08970=1082.463,-39.686,443.919,174.007,19.228,153.237
C08971=1082.469,-39.436,443.907,174.009,19.229,153.238
C08972=1082.475,-39.186,443.894,174.010,19.231,153.238
C08973=1082.482,-38.936,443.882,174.012,19.233,153.238
C08974=1082.487,-38.687,443.870,174.014,19.235,153.238
C08975=1082.493,-38.437,443.858,174.015,19.237,153.238
C08976=1082.499,-38.188,443.845,174.016,19.238,153.238
C08977=1082.505,-37.938,443.833,174.018,19.240,153.238
C08978=1082.511,-37.689,443.821,174.019,19.242,153.238
C08979=1082.517,-37.439,443.808,174.020,19.244,153.238
C08980=1082.522,-37.189,443.796,174.023,19.246,153.238
C08981=1082.528,-36.940,443.784,174.024,19.248,153.238
C08982=1082.534,-36.690,443.771,174.025,19.250,153.239
C08983=1082.540,-36.440,443.758,174.027,19.252,153.239
C08984=1082.546,-36.190,443.746,174.028,19.254,153.239
C08985=1082.552,-35.941,443.734,174.029,19.255,153.239
C08986=1082.557,-35.691,443.722,174.030,19.257,153.239
C08987=1082.563,-35.442,443.709,174.033,19.259,153.239
C08988=1082.569,-35.192,443.697,174.034,19.261,153.239
C08989=1082.575,-34.943,443.684,174.035,19.263,153.239
C08990=1082.581,-34.693,443.671,174.037,19.265,153.239
C08991=1082.587,-34.443,443.659,174.038,19.266,153.239
C08992=1082.593,-34.193,443.646,174.039,19.268,153.240
C08993=1082.599,-33.944,443.634,174.042,19.270,153.240
C08994=1082.605,-33.695,443.622,174.043,19.272,153.240
C08995=1082.611,-33.422,443.608,174.044,19.274,153.240
C08996=1082.618,-33.148,443.594,174.046,19.276,153.240
C08997=1082.624,-32.876,443.580,174.048,19.278,153.240
C08998=1082.630,-32.602,443.567,174.049,19.280,153.240
C08999=1082.637,-32.353,443.554,174.050,19.282,153.240
C09000=1082.642,-32.104,443.542,174.052,19.284,153.241
C09001=1082.648,-31.854,443.529,174.054,19.286,153.241
C09002=1082.654,-31.604,443.517,174.055,19.288,153.241
C09003=1082.660,-31.355,443.504,174.056,19.290,153.241
C09004=1082.666,-31.105,443.491,174.058,19.292,153.241
C09005=1082.672,-30.855,443.478,174.059,19.294,153.241
C09006=1082.677,-30.606,443.466,174.060,19.295,153.241
C09007=1082.683,-30.356,443.453,174.062,19.298,153.241
C09008=1082.689,-30.107,443.440,174.064,19.299,153.241
C09009=1082.695,-29.857,443.428,174.065,19.301,153.241
C09010=1082.701,-29.607,443.415,174.067,19.303,153.242
C09011=1082.707,-29.357,443.403,174.068,19.305,153.242
C09012=1082.713,-29.108,443.389,174.069,19.306,153.242
C09013=1082.719,-28.858,443.377,174.071,19.309,153.242
C09014=1082.725,-28.609,443.365,174.073,19.311,153.242
C09015=1082.731,-28.360,443.351,174.074,19.312,153.242
C09016=1082.737,-28.110,443.339,174.075,19.314,153.242
C09017=1082.743,-27.860,443.327,174.077,19.316,153.242
C09018=1082.749,-27.611,443.314,174.078,19.318,153.242
C09019=1082.756,-27.361,443.301,174.080,19.320,153.242
C09020=1082.761,-27.111,443.288,174.081,19.322,153.243
C09021=1082.767,-26.861,443.276,174.083,19.323,153.243
C09022=1082.773,-26.612,443.262,174.084,19.325,153.243
C09023=1082.778,-26.363,443.250,174.085,19.328,153.243
C09024=1082.784,-26.113,443.237,174.087,19.329,153.243
C09025=1082.790,-25.864,443.224,174.089,19.332,153.243
C09026=1082.796,-25.614,443.211,174.090,19.334,153.243
C09027=1082.802,-25.364,443.198,174.092,19.335,153.243
C09028=1082.808,-25.115,443.186,174.093,19.337,153.244
C09029=1082.813,-24.864,443.172,174.094,19.339,153.244
C09030=1082.819,-24.616,443.160,174.096,19.341,153.244
C09031=1082.825,-24.366,443.147,174.098,19.343,153.244
C09032=1082.831,-24.117,443.134,174.099,19.345,153.244
C09033=1082.837,-23.867,443.121,174.100,19.347,153.244
C09034=1082.843,-23.617,443.109,174.101,19.349,153.244
C09035=1082.848,-23.367,443.095,174.104,19.351,153.244
C09036=1082.854,-23.117,443.082,174.105,19.353,153.244
C09037=1082.861,-22.868,443.069,174.106,19.355,153.245
C09038=1082.867,-22.618,443.056,174.107,19.357,153.245
C09039=1082.873,-22.369,443.043,174.109,19.358,153.245
C09040=1082.878,-22.119,443.030,174.110,19.360,153.245
C09041=1082.884,-21.870,443.017,174.112,19.363,153.245
C09042=1082.889,-21.620,443.004,174.114,19.364,153.245
C09043=1082.896,-21.371,442.991,174.115,19.366,153.245
C09044=1082.902,-21.121,442.979,174.116,19.368,153.246
C09045=1082.907,-20.872,442.965,174.118,19.370,153.246
C09046=1082.913,-20.622,442.952,174.120,19.373,153.246
C09047=1082.919,-20.373,442.939,174.121,19.375,153.246
C09048=1082.925,-20.123,442.926,174.122,19.376,153.246
C09049=1082.931,-19.873,442.913,174.124,19.378,153.246
C09050=1082.936,-19.623,442.900,174.125,19.380,153.246
C09051=1082.943,-19.374,442.887,174.127,19.382,153.246
C09052=1082.949,-19.124,442.874,174.128,19.384,153.246
C09053=1082.955,-18.875,442.861,174.130,19.386,153.247
C09054=1082.960,-18.625,442.847,174.131,19.388,153.247
C09055=1082.966,-18.375,442.834,174.132,19.390,153.247
C09056=1082.972,-18.126,442.821,174.134,19.392,153.247
C09057=1082.978,-17.876,442.809,174.136,19.394,153.247
C09058=1082.985,-17.627,442.795,174.137,19.396,153.247
C09059=1082.991,-17.353,442.780,174.138,19.398,153.247
C09060=1082.997,-17.079,442.766,174.140,19.400,153.247
C09061=1083.004,-16.806,442.752,174.142,19.402,153.248
C09062=1083.010,-16.532,442.738,174.144,19.404,153.248
C09063=1083.016,-16.282,442.724,174.145,19.406,153.248
C09064=1083.022,-16.033,442.711,174.146,19.408,153.248
C09065=1083.028,-15.783,442.698,174.148,19.410,153.248
C09066=1083.034,-15.534,442.685,174.150,19.412,153.248
C09067=1083.040,-15.284,442.671,174.151,19.414,153.248
C09068=1083.045,-15.034,442.658,174.152,19.416,153.248
C09069=1083.052,-14.785,442.645,174.154,19.418,153.249
C09070=1083.057,-14.536,442.631,174.155,19.420,153.249
C09071=1083.063,-14.286,442.619,174.157,19.423,153.249
C09072=1083.069,-14.036,442.605,174.158,19.424,153.249
C09073=1083.075,-13.787,442.592,174.160,19.426,153.249
C09074=1083.080,-13.537,442.578,174.161,19.428,153.249
C09075=1083.086,-13.287,442.565,174.162,19.430,153.249
C09076=1083.092,-13.038,442.552,174.164,19.432,153.249
C09077=1083.098,-12.789,442.538,174.166,19.434,153.250
C09078=1083.104,-12.539,442.525,174.167,19.436,153.250
C09079=1083.109,-12.289,442.512,174.168,19.438,153.250
C09080=1083.115,-12.040,442.498,174.170,19.440,153.250
C09081=1083.121,-11.790,442.484,174.172,19.442,153.250
C09082=1083.127,-11.541,442.471,174.173,19.444,153.250
C09083=1083.132,-11.291,442.458,174.174,19.446,153.250
C09084=1083.138,-11.041,442.445,174.176,19.448,153.251
C09085=1083.145,-10.791,442.431,174.178,19.450,153.251
C09086=1083.151,-10.542,442.417,174.179,19.452,153.251
C09087=1083.156,-10.292,442.403,174.180,19.454,153.251
C09088=1083.162,-10.042,442.391,174.182,19.456,153.251
C09089=1083.168,-9.793,442.377,174.184,19.458,153.251
C09090=1083.174,-9.544,442.364,174.185,19.460,153.251
C09091=1083.179,-9.294,442.350,174.186,19.462,153.252
C09092=1083.186,-9.045,442.337,174.188,19.464,153.252
C09093=1083.191,-8.795,442.323,174.189,19.466,153.252
C09094=1083.197,-8.546,442.309,174.191,19.468,153.252
C09095=1083.202,-8.296,442.296,174.192,19.470,153.252
C09096=1083.209,-8.047,442.283,174.194,19.472,153.252
C09097=1083.215,-7.796,442.269,174.195,19.474,153.252
C09098=1083.221,-7.547,442.256,174.197,19.477,153.252
C09099=1083.226,-7.297,442.242,174.198,19.479,153.253
C09100=1083.233,-7.048,442.228,174.200,19.480,153.253
C09101=1083.238,-6.799,442.215,174.201,19.482,153.253
C09102=1083.244,-6.549,442.201,174.203,19.485,153.253
C09103=1083.250,-6.300,442.187,174.204,19.487,153.253
